(* IEC 61131-3 sources: com.logicals.lc3.webinar/usRTS_RPMControl_iSOC/src_FB_LIB_SAFE/Safe/PLCOpen, 23 files *)

(* ---- SF_MutingPar.iecst ---- *)
USING logicals.web.standard.safe;

NAMESPACE logicals.web.standard.safe
NAMESPACE plcopen

TYPE
	SF_MutingPar_State : UINT(
	/* Static Reset condition detected after FB activation in state 8401. */
	Reset_Error_1 := 16#C001,
	/* Static Reset condition detected in state 8402. */
	Reset_Error_2 := 16#C011,
	/* Error detected in muting sequence state 8000, 8010, 8310, 8020, 8040, 8030, 8330, 8110, 8410, 8120, 8140, 8130 or 8430. */
	Error_Muting_Sequence := 16#C004,
	/* DiscTime11_12, DiscTime21_22 or MaxMutingTime value out of range. */
	Parameter_Error := 16#C010,
	/* Timing error: Active muting time (when S_MutingActive = TRUE) exceeds MaxMutingTime. */
	Error_Timer_MaxMuting := 16#C020,
	/* Timing error: Discrepancy time for switching MutingSwitch11 and MutingSwitch12 > DiscTime11_12. */
	Error_Timer_MS11_12 := 16#C030,
	/* Timing error: Discrepancy time for switching MutingSwitch21 and MutingSwitch22 > DiscTime21_22. */
	Error_Timer_MS21_22 := 16#C040,
	/* Timing error: Discrepancy time for switching MutingSwitch21 and MutingSwitch22 > DiscTime21_22. */
	Idle := 16#0000,
	/* Muting not active and no safety demand from AOPD. If timers from subsequent muting are still running, they are stopped. */
	AOPD_Free := 16#8000,
	/* Function block has been activated. */
	Init := 16#8401,
	/* Safety demand detected by AOPD, muting not active. */
	Safety_Demand_AOPD := 16#8802,
	/* Safety demand or errors have been detected and are now cleared. Operator acknowledgment by Reset required. */
	Wait_for_Reset := 16#8402,
	/* Safety function activated. */
	Safe := 16#8002,
	/* Muting forward sequence is in starting phase after rising trigger of MutingSwitch 11.
	 * Monitoring of DiscTime11_12 is activated. Monitoring of MaxMutingTime is activated.
	 */
	Muting_Forward_Start_1 := 16#8010,
	/* Muting forward sequence is in starting phase after rising trigger of MutingSwitch 12. Monitoring of DiscTime11_12 is activated.
	 * Monitoring of MaxMutingTime is activated.
	 */
	Muting_Forward_Start_2 := 16#8310,
	/* Muting forward sequence is active either:
	 * - After rising trigger of the second entry MutingSwitch 12 or 11 has been detected.
	 * - When both MutingSwitch 11 and 12 have been actuated in the same cycle.
	 * Monitoring of DiscTime11_12 is stopped. Monitoring of MaxMutingTime is activated, when transition came directly from state 8000.
	 */
	Muting_Forward_Active_1 := 16#8020,
	/* Muting forward sequence is active. MutingSwitch21 is the first exit switch actuated. Monitoring of DiscTime21_22 is started. */
	Muting_Forward_Step_1 := 16#8030,
	/* Muting forward sequence is active. MutingSwitch22 is the first exit switch actuated. Monitoring of DiscTime21_22 is started. */
	Muting_Forward_Step_2 := 16#8330,
	/* Muting forward sequence is still active. Both MutingSwitch21 and 22 are actuated, the monitoring of DiscTime21_22 is stopped. */
	Muting_Forward_Active_2 := 16#8040,
	/* Muting backward sequence is in starting phase after rising trigger of MutingSwitch21.
	 * Monitoring of DiscTime21_22 is activated. Monitoring of MaxMutingTime is activated.
	 */
	Muting_Backward_Start_1 := 16#8110,
	/* Muting backward sequence is in starting phase after rising trigger of MutingSwitch22.
	 * Monitoring of DiscTime21_22 is activated. Monitoring of MaxMutingTime is activated.
	 */
	Muting_Backward_Start_2 := 16#8410,
	/* Muting backward sequence is active either:
	 * - After rising trigger of the second MutingSwitch 21 or 22 has been detected.
	 * - When both MutingSwitch 21 and 22 have been actuated in the same cycle.
	 * Monitoring of DiscTime21_22 is stopped. Monitoring of MaxMuting-Time is activated, when transition came directly from state 8000.
	 */
	Muting_Backward_Active_1 := 16#8120,
	/* Muting backward sequence is active. MutingSwitch11 is the first exit switch actuated. Monitoring of DiscTime11_12 is started. */
	Muting_Backward_Step_1 := 16#8130,
	/* Muting backward sequence is active. MutingSwitch12 is the first exit switch actuated. Monitoring of DiscTime11_12 is started. */
	Muting_Backward_Step_2 := 16#8430,
	/* Muting backward sequence is still active. Both exit switches MutingSwitch11 and 12 are actuated, the monitoring of DiscTime11_12 is stopped. */
	Muting_Backward_Active_2 := 16#8140
	);
END_TYPE

/* Muting is the intended suppression of the safety function. In this FB, parallel muting with four muting sensors is specified. */

FUNCTION_BLOCK SF_MutingPar
	{ altName:="SF_MutingPar"; bgColor:="Gold"; width:=360; }
	VAR_INPUT
		/* See Section 5.1.1 General Input Parameters */
		Activate : BOOL := FALSE;
		/* Variable.
		 * OSSD signal from AOPD.
		 * FALSE: Protection field interrupted.
		 * TRUE: Protection field not interrupted.
		 */
		S_AOPD_In : SAFEBOOL := SAFEBOOL_Constant#SAFEFALSE;
		/* Variable.
		 * Status of Muting sensor 11.
		 * FALSE: Muting sensor 11 not actuated.
		 * TRUE: Workpiece actuates muting sensor 11.
		 * Depending on the safety requirements it can be necessary to connect a SAFEBOOL.
		 */
		MutingSwitch11 : BOOL := FALSE;
		/* Variable.
		 * Status of Muting sensor 12.
		 * FALSE: Muting sensor 12 not actuated.
		 * TRUE: Workpiece actuates muting sensor 12.
		 * Depending on the safety requirements it can be necessary to connect a SAFEBOOL.
		 */
		MutingSwitch12 : BOOL := FALSE;
		/* Variable.
		 * Status of Muting sensor 21.
		 * FALSE: Muting sensor 21 not actuated.
		 * TRUE: Workpiece actuates muting sensor 21.
		 * Depending on the safety requirements it can be necessary to connect a SAFEBOOL.
		 */
		MutingSwitch21 : BOOL := FALSE;
		/* Variable.
		 * Status of Muting sensor 22.
		 * FALSE: Muting sensor 22 not actuated.
		 * TRUE: Workpiece actuates muting sensor 22.
		 * Depending on the safety requirements it can be necessary to connect a SAFEBOOL.
		 */
		MutingSwitch22 : BOOL := FALSE;
		/* Constant 0..4 s;
		 * Maximum discrepancy time for MutingSwitch11 and MutingSwitch12.
		 */
		DiscTime11_12 : TIME := T#0s;
		/* Constant 0..4 s;
		 * Maximum discrepancy time for MutingSwitch21 and MutingSwitch22.
		 */
		DiscTime21_22 : TIME := T#0s;
		/* Constant 0..120 min (application area specific);
		 * Maximum time for complete muting sequence, timer started when first 2 muting sensors are actuated.
		 */
		MaxMutingTime : TIME := T#0s;
		/* Variable or constant.
		 * Command by the control system that enables the start of the muting function when needed by the machine cycle.
		 * After the start of the muting function, this signal can be switched off.
		 * FALSE: Muting not enabled
		 * TRUE: Start of Muting function enabled
		 */
		MutingEnable : BOOL := FALSE;
		/* See Section 5.1.1 General Input Parameters */
		S_StartReset : SAFEBOOL := SAFEBOOL_Constant#SAFEFALSE;
		/* See Section 5.1.1 General Input Parameters */
		Reset : BOOL := FALSE;
	END_VAR
	VAR_OUTPUT
		/* See Section 5.1.2 General Output Parameters */
		Ready : BOOL := FALSE;
		/* Safety related output, indicates status of the muted guard.
		 * FALSE: AOPD protection field interrupted and muting not active.
		 * TRUE: AOPD protection field not interrupted or muting active.
		 */
		S_AOPD_Out : SAFEBOOL := SAFEBOOL_Constant#SAFEFALSE;
		/* Indicates status of Muting process.
		 * FALSE: Muting not active.
		 * TRUE: Muting active.
		 */
		S_MutingActive : SAFEBOOL := SAFEBOOL_Constant#SAFEFALSE;
		/* Optional. See 5.1.2 General Output Parameters */
		SafetyDemand : BOOL := FALSE;
		/* Optional. See 5.1.2 General Output Parameters */
		ResetRequest : BOOL := FALSE;
		/* See Section 5.1.2 General Output Parameters */
		Error : BOOL := FALSE;
		/* See Section 5.1.2 General Output Parameters */
		DiagCode : WORD := 16#000;
	END_VAR
	VAR
		/* ControlCode is used for state tracking */
		ControlCode : UINT := 16#0000;
		DiscTimer11_12 : TON;
		DiscTimer21_22 : TON;
		MaxMutingTimer : TON;
		R_Trig_Reset : R_TRIG;
		R_Trig_S11: R_TRIG;
		R_Trig_S12: R_TRIG;
		R_Trig_S21: R_TRIG;
		R_Trig_S22: R_TRIG;
		F_Trig_S11: F_TRIG;
		F_Trig_S12: F_TRIG;
		F_Trig_S21: F_TRIG;
		F_Trig_S22: F_TRIG;
	END_VAR

	R_Trig_Reset(Reset);
	R_Trig_S11(MutingSwitch11);
	R_Trig_S12(MutingSwitch12);
	R_Trig_S21(MutingSwitch21);
	R_Trig_S22(MutingSwitch22);
	F_Trig_S11(MutingSwitch11);
	F_Trig_S12(MutingSwitch12);
	F_Trig_S21(MutingSwitch21);
	F_Trig_S22(MutingSwitch22);

	IF(NOT Activate) THEN
		ControlCode := SF_MutingPar_State#Idle;
		DiagCode := TO_WORD(ControlCode);
	ELSE
		CASE TO_UINT(ControlCode) OF
			SF_MutingPar_State#Idle:
				/* IF(Activate) THEN - Active is always true here */
					ControlCode := SF_MutingPar_State#Init;
					DiagCode := TO_WORD(ControlCode);
			SF_MutingPar_State#Init:
				IF(Reset AND NOT R_Trig_Reset.Q) THEN
					ControlCode := SF_MutingPar_State#Reset_Error_1;
					DiagCode := TO_WORD(ControlCode);
				ELSIF(DiscTime11_12 > T#4s OR DiscTime11_12 < T#0s OR DiscTime21_22 > T#4s OR DiscTime21_22 < T#0s OR MaxMutingTime > T#120m OR MaxMutingTime < T#0m) THEN
					ControlCode := SF_MutingPar_State#Parameter_Error;
					DiagCode := TO_WORD(ControlCode);
				ELSIF(R_Trig_Reset.Q OR IS(S_StartReset)) THEN
					ControlCode := SF_MutingPar_State#Safe;
					DiagCode := TO_WORD(ControlCode);
				END_IF;
			SF_MutingPar_State#Reset_Error_1:
				IF(NOT Reset) THEN
					ControlCode := SF_MutingPar_State#Init;
					DiagCode := TO_WORD(ControlCode);
				END_IF;
			SF_MutingPar_State#Safe:
				IF(IS_NOT(S_AOPD_In)) THEN
					ControlCode := SF_MutingPar_State#Safety_Demand_AOPD;
					DiagCode := TO_WORD(ControlCode);
				/* ELSIF(IS(S_AOPD_In)) THEN */
				ELSE
					ControlCode := SF_MutingPar_State#AOPD_Free;
					DiagCode := TO_WORD(ControlCode);
				END_IF;
			SF_MutingPar_State#Safety_Demand_AOPD:
				IF(IS(S_AOPD_In)) THEN
					ControlCode := SF_MutingPar_State#Wait_for_Reset;
					DiagCode := TO_WORD(ControlCode);
				END_IF;
			SF_MutingPar_State#Wait_for_Reset:
				IF(Reset AND NOT R_Trig_Reset.Q) THEN
					ControlCode := SF_MutingPar_State#Reset_Error_2;
					DiagCode := TO_WORD(ControlCode);
				ELSIF(R_Trig_Reset.Q) THEN
					ControlCode := SF_MutingPar_State#Safe;
					DiagCode := TO_WORD(ControlCode);
				END_IF;
			SF_MutingPar_State#Reset_Error_2:
				IF(NOT Reset) THEN
					ControlCode := SF_MutingPar_State#Wait_for_Reset;
					DiagCode := TO_WORD(ControlCode);
				END_IF;
			SF_MutingPar_State#AOPD_Free:
				/* MutingEnable missing when muting sequence starts */
				IF(NOT MutingEnable) THEN
					IF((R_Trig_S11.Q AND NOT MutingSwitch12 AND NOT MutingSwitch21 AND NOT MutingSwitch22) OR
						(NOT MutingSwitch11 AND R_Trig_S12.Q AND NOT MutingSwitch21 AND NOT MutingSwitch22) OR
						(NOT MutingSwitch22 AND R_Trig_S21.Q AND NOT MutingSwitch11 AND NOT MutingSwitch12) OR
						(R_Trig_S22.Q AND NOT MutingSwitch21 AND NOT MutingSwitch11 AND NOT MutingSwitch12) OR
						(R_Trig_S11.Q AND R_Trig_S12.Q AND NOT MutingSwitch21 AND NOT MutingSwitch22) OR
						(R_Trig_S21.Q AND R_Trig_S22.Q AND NOT MutingSwitch11 AND NOT MutingSwitch12)) THEN
							ControlCode := SF_MutingPar_State#Error_Muting_Sequence;
							DiagCode := TO_WORD(SF_MutingPar_State#Error_Muting_Sequence + 16#0F00 + MutingParGetErrorStateOfMutingSensors(MutingSwitch11, MutingSwitch12, MutingSwitch21, MutingSwitch22));
					END_IF;
				/* wrong muting sequence */
				ELSIF((MutingSwitch11 OR MutingSwitch12) AND (MutingSwitch21 OR MutingSwitch22)) OR
					(R_Trig_S11.Q AND MutingSwitch12 AND NOT R_Trig_S12.Q) OR
					(R_Trig_S12.Q AND MutingSwitch11 AND NOT R_Trig_S11.Q) OR
					(R_Trig_S21.Q AND MutingSwitch22 AND NOT R_Trig_S22.Q) OR
					(R_Trig_S22.Q AND MutingSwitch21 AND NOT R_Trig_S21.Q) OR
					((MutingSwitch11 AND NOT R_Trig_S11.Q) AND (MutingSwitch12 AND NOT R_Trig_S12.Q)) OR
					((MutingSwitch21 AND NOT R_Trig_S21.Q) AND (MutingSwitch22 AND NOT R_Trig_S22.Q)) THEN
						ControlCode := SF_MutingPar_State#Error_Muting_Sequence;
						DiagCode := TO_WORD(SF_MutingPar_State#Error_Muting_Sequence + MutingParGetErrorStateOfMutingSensors(MutingSwitch11, MutingSwitch12, MutingSwitch21, MutingSwitch22));
				ELSIF(IS_NOT(S_AOPD_In)) THEN
					ControlCode := SF_MutingPar_State#Safety_Demand_AOPD;
					DiagCode := TO_WORD(ControlCode);
				ELSIF(MutingEnable AND (R_Trig_S11.Q AND NOT MutingSwitch12 AND NOT MutingSwitch21 AND NOT MutingSwitch22)) THEN
					ControlCode := SF_MutingPar_State#Muting_Forward_Start_1;
					DiagCode := TO_WORD(ControlCode);
				ELSIF(MutingEnable AND (NOT MutingSwitch11 AND R_Trig_S12.Q AND NOT MutingSwitch21 AND NOT MutingSwitch22)) THEN
					ControlCode := SF_MutingPar_State#Muting_Forward_Start_2;
					DiagCode := TO_WORD(ControlCode);
				ELSIF(MutingEnable AND (NOT MutingSwitch22 AND R_Trig_S21.Q AND NOT MutingSwitch11 AND NOT MutingSwitch12)) THEN
					ControlCode := SF_MutingPar_State#Muting_Backward_Start_1;
					DiagCode := TO_WORD(ControlCode);
				ELSIF(MutingEnable AND (R_Trig_S22.Q AND NOT MutingSwitch21 AND NOT MutingSwitch11 AND NOT MutingSwitch12)) THEN
					ControlCode := SF_MutingPar_State#Muting_Backward_Start_2;
					DiagCode := TO_WORD(ControlCode);
				ELSIF(MutingEnable AND (R_Trig_S11.Q AND R_Trig_S12.Q AND NOT MutingSwitch21 AND NOT MutingSwitch22)) THEN
					ControlCode := SF_MutingPar_State#Muting_Forward_Active_1;
					DiagCode := TO_WORD(ControlCode);
				ELSIF(MutingEnable AND (R_Trig_S21.Q AND R_Trig_S22.Q AND NOT MutingSwitch11 AND NOT MutingSwitch12)) THEN
					ControlCode := SF_MutingPar_State#Muting_Backward_Active_1;
					DiagCode := TO_WORD(ControlCode);
				END_IF;
			SF_MutingPar_State#Muting_Forward_Start_1:
				DiscTimer11_12();
				MaxMutingTimer();
				IF(NOT MutingEnable) THEN
					ControlCode := SF_MutingPar_State#Error_Muting_Sequence;
					DiagCode := TO_WORD(SF_MutingPar_State#Error_Muting_Sequence + 16#0F00 + MutingParGetErrorStateOfMutingSensors(MutingSwitch11, MutingSwitch12, MutingSwitch21, MutingSwitch22));
				ELSIF(NOT MutingSwitch11 OR MutingSwitch21 OR MutingSwitch22) THEN
					ControlCode := SF_MutingPar_State#Error_Muting_Sequence;
					DiagCode := TO_WORD(SF_MutingPar_State#Error_Muting_Sequence + 16#0100 + MutingParGetErrorStateOfMutingSensors(MutingSwitch11, MutingSwitch12, MutingSwitch21, MutingSwitch22));
				ELSIF(DiscTimer11_12.Q) THEN
					ControlCode := SF_MutingPar_State#Error_Timer_MS11_12;
					DiagCode := TO_WORD(ControlCode);
				ELSIF(MaxMutingTimer.Q) THEN
					ControlCode := SF_MutingPar_State#Error_Timer_MaxMuting;
					DiagCode := TO_WORD(ControlCode);
				ELSIF(IS_NOT(S_AOPD_In)) THEN
					ControlCode := SF_MutingPar_State#Safety_Demand_AOPD;
					DiagCode := TO_WORD(ControlCode);
				ELSIF(MutingEnable AND(MutingSwitch11 AND R_Trig_S12.Q AND NOT MutingSwitch21 AND NOT MutingSwitch22)) THEN
					ControlCode := SF_MutingPar_State#Muting_Forward_Active_1;
					DiagCode := TO_WORD(ControlCode);
				END_IF;
			SF_MutingPar_State#Muting_Forward_Start_2:
				DiscTimer11_12();
				MaxMutingTimer();
				IF(NOT MutingEnable) THEN
					ControlCode := SF_MutingPar_State#Error_Muting_Sequence;
					DiagCode := TO_WORD(SF_MutingPar_State#Error_Muting_Sequence + 16#0F00 + MutingParGetErrorStateOfMutingSensors(MutingSwitch11, MutingSwitch12, MutingSwitch21, MutingSwitch22));
				ELSIF(NOT MutingSwitch12 OR MutingSwitch21 OR MutingSwitch22) THEN
					ControlCode := SF_MutingPar_State#Error_Muting_Sequence;
					DiagCode := TO_WORD(SF_MutingPar_State#Error_Muting_Sequence + 16#0200 + MutingParGetErrorStateOfMutingSensors(MutingSwitch11, MutingSwitch12, MutingSwitch21, MutingSwitch22));
				ELSIF(DiscTimer11_12.Q) THEN
					ControlCode := SF_MutingPar_State#Error_Timer_MS11_12;
					DiagCode := TO_WORD(ControlCode);
				ELSIF(MaxMutingTimer.Q) THEN
					ControlCode := SF_MutingPar_State#Error_Timer_MaxMuting;
					DiagCode := TO_WORD(ControlCode);
				ELSIF(IS_NOT(S_AOPD_In)) THEN
					ControlCode := SF_MutingPar_State#Safety_Demand_AOPD;
					DiagCode := TO_WORD(ControlCode);
				ELSIF(R_Trig_S11.Q AND MutingSwitch12 AND NOT MutingSwitch21 AND NOT MutingSwitch22) THEN
					ControlCode := SF_MutingPar_State#Muting_Forward_Active_1;
					DiagCode := TO_WORD(ControlCode);
				END_IF;
			SF_MutingPar_State#Muting_Backward_Start_1:
				DiscTimer21_22();
				MaxMutingTimer();
				IF(NOT MutingEnable) THEN
					ControlCode := SF_MutingPar_State#Error_Muting_Sequence;
					DiagCode := TO_WORD(SF_MutingPar_State#Error_Muting_Sequence + 16#0F00 + MutingParGetErrorStateOfMutingSensors(MutingSwitch11, MutingSwitch12, MutingSwitch21, MutingSwitch22));
				ELSIF(MutingSwitch11 OR MutingSwitch12 OR NOT MutingSwitch21) THEN
					ControlCode := SF_MutingPar_State#Error_Muting_Sequence;
					DiagCode := TO_WORD(SF_MutingPar_State#Error_Muting_Sequence + 16#0700 + MutingParGetErrorStateOfMutingSensors(MutingSwitch11, MutingSwitch12, MutingSwitch21, MutingSwitch22));
				ELSIF(DiscTimer21_22.Q) THEN
					ControlCode := SF_MutingPar_State#Error_Timer_MS21_22;
					DiagCode := TO_WORD(ControlCode);
				ELSIF(MaxMutingTimer.Q) THEN
					ControlCode := SF_MutingPar_State#Error_Timer_MaxMuting;
					DiagCode := TO_WORD(ControlCode);
				ELSIF(IS_NOT(S_AOPD_In)) THEN
					ControlCode := SF_MutingPar_State#Safety_Demand_AOPD;
					DiagCode := TO_WORD(ControlCode);
				ELSIF(MutingEnable AND (MutingSwitch21 AND R_Trig_S22.Q AND NOT MutingSwitch11 AND NOT MutingSwitch12)) THEN
					ControlCode := SF_MutingPar_State#Muting_Backward_Active_1;
					DiagCode := TO_WORD(ControlCode);
				END_IF;
			SF_MutingPar_State#Muting_Backward_Start_2:
				DiscTimer21_22();
				MaxMutingTimer();
				IF(NOT MutingEnable) THEN
					ControlCode := SF_MutingPar_State#Error_Muting_Sequence;
					DiagCode := TO_WORD(SF_MutingPar_State#Error_Muting_Sequence + 16#0F00 + MutingParGetErrorStateOfMutingSensors(MutingSwitch11, MutingSwitch12, MutingSwitch21, MutingSwitch22));
				ELSIF(MutingSwitch11 OR MutingSwitch12 OR NOT MutingSwitch22) THEN
					ControlCode := SF_MutingPar_State#Error_Muting_Sequence;
					DiagCode := TO_WORD(SF_MutingPar_State#Error_Muting_Sequence + 16#0800 + MutingParGetErrorStateOfMutingSensors(MutingSwitch11, MutingSwitch12, MutingSwitch21, MutingSwitch22));
				ELSIF(DiscTimer21_22.Q) THEN
					ControlCode := SF_MutingPar_State#Error_Timer_MS21_22;
					DiagCode := TO_WORD(ControlCode);
				ELSIF(MaxMutingTimer.Q) THEN
					ControlCode := SF_MutingPar_State#Error_Timer_MaxMuting;
					DiagCode := TO_WORD(ControlCode);
				ELSIF(IS_NOT(S_AOPD_In)) THEN
					ControlCode := SF_MutingPar_State#Safety_Demand_AOPD;
					DiagCode := TO_WORD(ControlCode);
				ELSIF(MutingEnable AND (R_Trig_S21.Q AND MutingSwitch22 AND NOT MutingSwitch11 AND NOT MutingSwitch12)) THEN
					ControlCode := SF_MutingPar_State#Muting_Backward_Active_1;
					DiagCode := TO_WORD(ControlCode);
				END_IF;
			SF_MutingPar_State#Muting_Forward_Active_1:
				MaxMutingTimer();
				IF(NOT MutingSwitch11 OR NOT MutingSwitch12) THEN
					ControlCode := SF_MutingPar_State#Error_Muting_Sequence;
					DiagCode := TO_WORD(SF_MutingPar_State#Error_Muting_Sequence + 16#0300 + MutingParGetErrorStateOfMutingSensors(MutingSwitch11, MutingSwitch12, MutingSwitch21, MutingSwitch22));
				ELSIF(MaxMutingTimer.Q) THEN
					ControlCode := SF_MutingPar_State#Error_Timer_MaxMuting;
					DiagCode := TO_WORD(ControlCode);
				ELSIF(MutingSwitch11 AND MutingSwitch12 AND MutingSwitch21 AND MutingSwitch22) THEN
					ControlCode := SF_MutingPar_State#Muting_Forward_Active_2;
					DiagCode := TO_WORD(ControlCode);
				ELSIF(MutingSwitch11 AND MutingSwitch12 AND R_Trig_S21.Q AND NOT MutingSwitch22) THEN
					ControlCode := SF_MutingPar_State#Muting_Forward_Step_1;
					DiagCode := TO_WORD(ControlCode);
				ELSIF(MutingSwitch11 AND MutingSwitch12 AND NOT MutingSwitch21 AND R_Trig_S22.Q) THEN
					ControlCode := SF_MutingPar_State#Muting_Forward_Step_2;
					DiagCode := TO_WORD(ControlCode);
				END_IF;
			SF_MutingPar_State#Muting_Forward_Step_1:
				DiscTimer21_22();
				MaxMutingTimer();
				IF(NOT MutingSwitch11 OR NOT MutingSwitch12 OR NOT MutingSwitch21) THEN
					ControlCode := SF_MutingPar_State#Error_Muting_Sequence;
					DiagCode := TO_WORD(SF_MutingPar_State#Error_Muting_Sequence + 16#0400 + MutingParGetErrorStateOfMutingSensors(MutingSwitch11, MutingSwitch12, MutingSwitch21, MutingSwitch22));
				ELSIF(DiscTimer21_22.Q) THEN
					ControlCode := SF_MutingPar_State#Error_Timer_MS21_22;
					DiagCode := TO_WORD(ControlCode);
				ELSIF(MaxMutingTimer.Q) THEN
					ControlCode := SF_MutingPar_State#Error_Timer_MaxMuting;
					DiagCode := TO_WORD(ControlCode);
				ELSIF(MutingSwitch11 AND MutingSwitch12 AND MutingSwitch21 AND R_Trig_S22.Q) THEN
					ControlCode := SF_MutingPar_State#Muting_Forward_Active_2;
					DiagCode := TO_WORD(ControlCode);
				END_IF;
			SF_MutingPar_State#Muting_Forward_Step_2:
				DiscTimer21_22();
				MaxMutingTimer();
				IF(NOT MutingSwitch11 OR NOT MutingSwitch12 OR NOT MutingSwitch22) THEN
					ControlCode := SF_MutingPar_State#Error_Muting_Sequence;
					DiagCode := TO_WORD(SF_MutingPar_State#Error_Muting_Sequence + 16#0500 + MutingParGetErrorStateOfMutingSensors(MutingSwitch11, MutingSwitch12, MutingSwitch21, MutingSwitch22));
				ELSIF(DiscTimer21_22.Q) THEN
					ControlCode := SF_MutingPar_State#Error_Timer_MS21_22;
					DiagCode := TO_WORD(ControlCode);
				ELSIF(MaxMutingTimer.Q) THEN
					ControlCode := SF_MutingPar_State#Error_Timer_MaxMuting;
					DiagCode := TO_WORD(ControlCode);
				ELSIF(MutingSwitch11 AND MutingSwitch12 AND R_Trig_S21.Q AND MutingSwitch22) THEN
					ControlCode := SF_MutingPar_State#Muting_Forward_Active_2;
					DiagCode := TO_WORD(ControlCode);
				END_IF;
			SF_MutingPar_State#Muting_Forward_Active_2:
				MaxMutingTimer();
				IF(R_Trig_S11.Q OR R_Trig_S12.Q OR R_Trig_S21.Q OR R_Trig_S22.Q) OR
					((MutingSwitch11 OR MutingSwitch12) AND (F_Trig_S21.Q OR F_Trig_S22.Q)) OR
					((F_Trig_S11.Q OR F_Trig_S12.Q) AND (F_Trig_S21.Q OR F_Trig_S22.Q)) THEN
						ControlCode := SF_MutingPar_State#Error_Muting_Sequence;
						DiagCode := TO_WORD(SF_MutingPar_State#Error_Muting_Sequence + 16#0600 + MutingParGetErrorStateOfMutingSensors(MutingSwitch11, MutingSwitch12, MutingSwitch21, MutingSwitch22));
				ELSIF(MaxMutingTimer.Q) THEN
					ControlCode := SF_MutingPar_State#Error_Timer_MaxMuting;
					DiagCode := TO_WORD(ControlCode);
				ELSIF(NOT MutingSwitch11 AND NOT MutingSwitch12) AND (F_Trig_S21.Q OR F_Trig_S22.Q) THEN
					ControlCode := SF_MutingPar_State#AOPD_Free;
					DiagCode := TO_WORD(ControlCode);
				END_IF;
			SF_MutingPar_State#Muting_Backward_Active_1:
				MaxMutingTimer();
				IF(NOT MutingSwitch21 OR NOT MutingSwitch22) THEN
					ControlCode := SF_MutingPar_State#Error_Muting_Sequence;
					DiagCode := TO_WORD(SF_MutingPar_State#Error_Muting_Sequence + 16#0900 + MutingParGetErrorStateOfMutingSensors(MutingSwitch11, MutingSwitch12, MutingSwitch21, MutingSwitch22));
				ELSIF(MaxMutingTimer.Q) THEN
					ControlCode := SF_MutingPar_State#Error_Timer_MaxMuting;
					DiagCode := TO_WORD(ControlCode);
				ELSIF(MutingSwitch11 AND MutingSwitch12 AND MutingSwitch21 AND MutingSwitch22) THEN
					ControlCode := SF_MutingPar_State#Muting_Backward_Active_2;
					DiagCode := TO_WORD(ControlCode);
				ELSIF(MutingSwitch21 AND MutingSwitch22 AND R_Trig_S11.Q AND NOT MutingSwitch12) THEN
					ControlCode := SF_MutingPar_State#Muting_Backward_Step_1;
					DiagCode := TO_WORD(ControlCode);
				ELSIF(MutingSwitch21 AND MutingSwitch22 AND NOT MutingSwitch11 AND R_Trig_S12.Q) THEN
					ControlCode := SF_MutingPar_State#Muting_Backward_Step_2;
					DiagCode := TO_WORD(ControlCode);
				END_IF;
			SF_MutingPar_State#Muting_Backward_Step_1:
				MaxMutingTimer();
				DiscTimer11_12();
				IF(NOT MutingSwitch21 OR NOT MutingSwitch22 OR NOT MutingSwitch11) THEN
					ControlCode := SF_MutingPar_State#Error_Muting_Sequence;
					DiagCode := TO_WORD(SF_MutingPar_State#Error_Muting_Sequence + 16#0A00 + MutingParGetErrorStateOfMutingSensors(MutingSwitch11, MutingSwitch12, MutingSwitch21, MutingSwitch22));
				ELSIF(DiscTimer11_12.Q) THEN
					ControlCode := SF_MutingPar_State#Error_Timer_MS11_12;
					DiagCode := TO_WORD(ControlCode);
				ELSIF(MaxMutingTimer.Q) THEN
					ControlCode := SF_MutingPar_State#Error_Timer_MaxMuting;
					DiagCode := TO_WORD(ControlCode);
				ELSIF(MutingSwitch21 AND MutingSwitch22 AND MutingSwitch11 AND R_Trig_S12.Q) THEN
					ControlCode := SF_MutingPar_State#Muting_Backward_Active_2;
					DiagCode := TO_WORD(ControlCode);
				END_IF;
			SF_MutingPar_State#Muting_Backward_Step_2:
				MaxMutingTimer();
				DiscTimer11_12();
				IF(NOT MutingSwitch21 OR NOT MutingSwitch22 OR NOT MutingSwitch12) THEN
					ControlCode := SF_MutingPar_State#Error_Muting_Sequence;
					DiagCode := TO_WORD(SF_MutingPar_State#Error_Muting_Sequence + 16#0B00 + MutingParGetErrorStateOfMutingSensors(MutingSwitch11, MutingSwitch12, MutingSwitch21, MutingSwitch22));
				ELSIF(DiscTimer11_12.Q) THEN
					ControlCode := SF_MutingPar_State#Error_Timer_MS11_12;
					DiagCode := TO_WORD(ControlCode);
				ELSIF(MaxMutingTimer.Q) THEN
					ControlCode := SF_MutingPar_State#Error_Timer_MaxMuting;
					DiagCode := TO_WORD(ControlCode);
				ELSIF(MutingSwitch21 AND MutingSwitch22 AND R_Trig_S11.Q AND MutingSwitch12) THEN
					ControlCode := SF_MutingPar_State#Muting_Backward_Active_2;
					DiagCode := TO_WORD(ControlCode);
				END_IF;
			SF_MutingPar_State#Muting_Backward_Active_2:
				MaxMutingTimer();
				IF(R_Trig_S11.Q OR R_Trig_S12.Q OR R_Trig_S21.Q OR R_Trig_S22.Q) OR
					((MutingSwitch21 OR MutingSwitch22) AND (F_Trig_S11.Q OR F_Trig_S12.Q)) OR
					((F_Trig_S11.Q OR F_Trig_S12.Q) AND (F_Trig_S21.Q OR F_Trig_S22.Q)) THEN
						ControlCode := SF_MutingPar_State#Error_Muting_Sequence;
						DiagCode := TO_WORD(SF_MutingPar_State#Error_Muting_Sequence + 16#0C00 + MutingParGetErrorStateOfMutingSensors(MutingSwitch11, MutingSwitch12, MutingSwitch21, MutingSwitch22));
				ELSIF(MaxMutingTimer.Q) THEN
					ControlCode := SF_MutingPar_State#Error_Timer_MaxMuting;
					DiagCode := TO_WORD(ControlCode);
				ELSIF(NOT MutingSwitch21 AND NOT MutingSwitch22 AND(F_Trig_S11.Q OR F_Trig_S12.Q)) THEN
					ControlCode := SF_MutingPar_State#AOPD_Free;
					DiagCode := TO_WORD(ControlCode);
				END_IF;
			SF_MutingPar_State#Error_Timer_MaxMuting,
			SF_MutingPar_State#Error_Timer_MS11_12,
			SF_MutingPar_State#Error_Timer_MS21_22:
				IF(NOT(MutingSwitch11 OR MutingSwitch12 OR MutingSwitch21 OR MutingSwitch22)) THEN
					ControlCode := SF_MutingPar_State#Wait_for_Reset;
					DiagCode := TO_WORD(ControlCode);
				END_IF;
			ELSE
				ENO := FALSE;
		END_CASE;
	END_IF;

	CASE TO_UINT(ControlCode) OF
		SF_MutingPar_State#Reset_Error_1,
		SF_MutingPar_State#Reset_Error_2,
		SF_MutingPar_State#Parameter_Error,
		SF_MutingPar_State#Error_Timer_MaxMuting,
		SF_MutingPar_State#Error_Timer_MS11_12,
		SF_MutingPar_State#Error_Timer_MS21_22:
			DiscTimer11_12(IN := FALSE);
			DiscTimer21_22(IN := FALSE);
			MaxMutingTimer(IN := FALSE);
			Ready := TRUE;
			S_AOPD_Out := SAFEBOOL_Constant#SAFEFALSE;
			S_MutingActive := SAFEBOOL_Constant#SAFEFALSE;
			SafetyDemand := FALSE;
			ResetRequest := FALSE;
			Error := TRUE;
		SF_MutingPar_State#Error_Muting_Sequence:
			DiscTimer11_12(IN := FALSE);
			DiscTimer21_22(IN := FALSE);
			MaxMutingTimer(IN := FALSE);
			Ready := TRUE;
			S_AOPD_Out := SAFEBOOL_Constant#SAFEFALSE;
			S_MutingActive := SAFEBOOL_Constant#SAFEFALSE;
			SafetyDemand := FALSE;
			ResetRequest := FALSE;
			Error := TRUE;
		SF_MutingPar_State#Idle:
			DiscTimer11_12(IN := FALSE);
			DiscTimer21_22(IN := FALSE);
			MaxMutingTimer(IN := FALSE);
			Ready := FALSE;
			S_AOPD_Out := SAFEBOOL_Constant#SAFEFALSE;
			S_MutingActive := SAFEBOOL_Constant#SAFEFALSE;
			SafetyDemand := FALSE;
			ResetRequest := FALSE;
			Error := FALSE;
		SF_MutingPar_State#AOPD_Free:
			DiscTimer11_12(IN := FALSE);
			DiscTimer21_22(IN := FALSE);
			MaxMutingTimer(IN := FALSE);
			Ready := TRUE;
			S_AOPD_Out := SAFEBOOL_Constant#SAFETRUE;
			S_MutingActive := SAFEBOOL_Constant#SAFEFALSE;
			SafetyDemand := FALSE;
			ResetRequest := FALSE;
			Error := FALSE;
		SF_MutingPar_State#Muting_Forward_Start_1,
		SF_MutingPar_State#Muting_Forward_Start_2:
			DiscTimer11_12(IN := TRUE, PT := DiscTime11_12);
			DiscTimer21_22(IN := FALSE);
			MaxMutingTimer(IN := TRUE, PT := MaxMutingTime);
			Ready := TRUE;
			S_AOPD_Out := SAFEBOOL_Constant#SAFETRUE;
			S_MutingActive := SAFEBOOL_Constant#SAFEFALSE;
			SafetyDemand := FALSE;
			ResetRequest := FALSE;
			Error := FALSE;
		SF_MutingPar_State#Muting_Backward_Start_1,
		SF_MutingPar_State#Muting_Backward_Start_2:
			DiscTimer11_12(IN := FALSE);
			DiscTimer21_22(IN := TRUE, PT := DiscTime21_22);
			MaxMutingTimer(IN := TRUE, PT := MaxMutingTime);
			Ready := TRUE;
			S_AOPD_Out := SAFEBOOL_Constant#SAFETRUE;
			S_MutingActive := SAFEBOOL_Constant#SAFEFALSE;
			SafetyDemand := FALSE;
			ResetRequest := FALSE;
			Error := FALSE;
		SF_MutingPar_State#Init,
		SF_MutingPar_State#Wait_for_Reset:
			DiscTimer11_12(IN := FALSE);
			DiscTimer21_22(IN := FALSE);
			MaxMutingTimer(IN := FALSE);
			Ready := TRUE;
			S_AOPD_Out := SAFEBOOL_Constant#SAFEFALSE;
			S_MutingActive := SAFEBOOL_Constant#SAFEFALSE;
			SafetyDemand := FALSE;
			ResetRequest := TRUE;
			Error := FALSE;
		SF_MutingPar_State#Safety_Demand_AOPD:
			DiscTimer11_12(IN := FALSE);
			DiscTimer21_22(IN := FALSE);
			MaxMutingTimer(IN := FALSE);
			Ready := TRUE;
			S_AOPD_Out := SAFEBOOL_Constant#SAFEFALSE;
			S_MutingActive := SAFEBOOL_Constant#SAFEFALSE;
			SafetyDemand := TRUE;
			ResetRequest := FALSE;
			Error := FALSE;
		SF_MutingPar_State#Safe:
			DiscTimer11_12(IN := FALSE);
			DiscTimer21_22(IN := FALSE);
			MaxMutingTimer(IN := FALSE);
			Ready := TRUE;
			S_AOPD_Out := SAFEBOOL_Constant#SAFEFALSE;
			S_MutingActive := SAFEBOOL_Constant#SAFEFALSE;
			SafetyDemand := FALSE;
			ResetRequest := FALSE;
			Error := FALSE;
		SF_MutingPar_State#Muting_Backward_Active_1:
			DiscTimer11_12(IN := FALSE);
			DiscTimer21_22(IN := FALSE);
			IF(MutingEnable AND (R_Trig_S21.Q AND R_Trig_S22.Q AND NOT MutingSwitch11 AND NOT MutingSwitch12)) THEN
				MaxMutingTimer(IN := TRUE, PT:= MaxMutingTime);
			END_IF;
			Ready := TRUE;
			S_AOPD_Out := SAFEBOOL_Constant#SAFETRUE;
			S_MutingActive := SAFEBOOL_Constant#SAFETRUE;
			SafetyDemand := FALSE;
			ResetRequest := FALSE;
			Error := FALSE;
		SF_MutingPar_State#Muting_Backward_Step_1,
		SF_MutingPar_State#Muting_Backward_Step_2:
			DiscTimer11_12(IN := TRUE, PT := DiscTime11_12);
			DiscTimer21_22(IN := FALSE);
			Ready := TRUE;
			S_AOPD_Out := SAFEBOOL_Constant#SAFETRUE;
			S_MutingActive := SAFEBOOL_Constant#SAFETRUE;
			SafetyDemand := FALSE;
			ResetRequest := FALSE;
			Error := FALSE;
		SF_MutingPar_State#Muting_Backward_Active_2:
			DiscTimer11_12(IN := FALSE);
			DiscTimer21_22(IN := FALSE);
			Ready := TRUE;
			S_AOPD_Out := SAFEBOOL_Constant#SAFETRUE;
			S_MutingActive := SAFEBOOL_Constant#SAFETRUE;
			SafetyDemand := FALSE;
			ResetRequest := FALSE;
			Error := FALSE;
		SF_MutingPar_State#Muting_Forward_Active_1:
			DiscTimer11_12(IN := FALSE);
			DiscTimer21_22(IN := FALSE);
			IF(MutingEnable AND (R_Trig_S11.Q AND R_Trig_S12.Q AND NOT MutingSwitch21 AND NOT MutingSwitch22)) THEN
				MaxMutingTimer(IN := TRUE, PT:= MaxMutingTime);
			END_IF;
			Ready := TRUE;
			S_AOPD_Out := SAFEBOOL_Constant#SAFETRUE;
			S_MutingActive := SAFEBOOL_Constant#SAFETRUE;
			SafetyDemand := FALSE;
			ResetRequest := FALSE;
			Error := FALSE;
		SF_MutingPar_State#Muting_Forward_Step_1,
		SF_MutingPar_State#Muting_Forward_Step_2:
			DiscTimer11_12(IN := FALSE);
			DiscTimer21_22(IN := TRUE, PT := DiscTime21_22);
			Ready := TRUE;
			S_AOPD_Out := SAFEBOOL_Constant#SAFETRUE;
			S_MutingActive := SAFEBOOL_Constant#SAFETRUE;
			SafetyDemand := FALSE;
			ResetRequest := FALSE;
			Error := FALSE;
		SF_MutingPar_State#Muting_Forward_Active_2:
			DiscTimer11_12(IN := FALSE);
			DiscTimer21_22(IN := FALSE);
			Ready := TRUE;
			S_AOPD_Out := SAFEBOOL_Constant#SAFETRUE;
			S_MutingActive := SAFEBOOL_Constant#SAFETRUE;
			SafetyDemand := FALSE;
			ResetRequest := FALSE;
			Error := FALSE;
		ELSE
			ENO := FALSE;
	END_CASE;

	ENO := ENO AND CheckSAFEBOOL(S_AOPD_In) AND CheckSAFEBOOL(S_StartReset);

END_FUNCTION_BLOCK

FUNCTION MutingParGetErrorStateOfMutingSensors : UINT
	VAR_INPUT
		MS_11 : BOOL;
		MS_12 : BOOL;
		MS_21 : BOOL;
		MS_22 : BOOL;
	END_VAR

	VAR
		Result : UINT;
	END_VAR

	IF(MS_11) THEN
		Result := Result + 16#0010;
	END_IF;
	IF(MS_12) THEN
		Result := Result + 16#0020;
	END_IF;
	IF(MS_21) THEN
		Result := Result + 16#0040;
	END_IF;
	IF(MS_22) THEN
		Result := Result + 16#0080;
	END_IF;

	MutingParGetErrorStateOfMutingSensors := Result;

END_FUNCTION

END_NAMESPACE
END_NAMESPACE

(* ---- SF_Antivalent.iecst ---- *)
USING logicals.web.standard.safe;

NAMESPACE logicals.web.standard.safe
NAMESPACE plcopen

TYPE
	SF_Antivalent_State : UINT(
	/* Discrepancy time elapsed in state 8802. */
	Error_1 := 16#C010,
	/* Discrepancy time elapsed in state 8804. */
	Error_2 := 16#C020,
	/* Discrepancy time elapsed in state 8806. */
	Error_3 := 16#C030,
	/* The function block is not active (initial state). */
	Idle := 16#0000,
	/* An activation has been detected by the FB and the FB is now activated. */
	Init := 16#8801,
	/* The inputs switched to the Active state in antivalent mode. */
	Safety_Output_Enabled := 16#8000,
	/* ChannelNC has been switched to TRUE - waiting for ChannelNO to be switched to FALSE; discrepancy timer started. */
	Wait_for_NO := 16#8802,
	/* ChannelNO has been switched to FALSE - waiting for ChannelNC to be switched to TRUE; discrepancy timer started. */
	Wait_for_NC := 16#8804,
	/* One channel has been switched to inactive; waiting for the second channel to be switched to inactive too. */
	From_Active_Wait := 16#8806
	);
END_TYPE

/*
 * This function block converts two antivalent SAFEBOOL inputs (NO/NC pair) to one SAFEBOOL output with discrepancy time monitoring.
 * This FB should not be used stand-alone since it has no restart interlock.
 * It is required to connect the output to other safety related functionalities.
 */
FUNCTION_BLOCK SF_Antivalent
	{ altName:="SF_Antivalent"; bgColor:="Gold"; width:=380; }
	VAR_INPUT
		/* See Section 5.1.1 General Input Parameters */
		Activate : BOOL := FALSE;
		/* Variable. NC stands for Normally Closed.
		 * Input for NC connection.
		 * FALSE: NC contact open.
		 * TRUE: NC contact closed. */
		S_ChannelNC : SAFEBOOL := SAFEBOOL_Constant#SAFEFALSE;
		/* Variable. NO stands for Normally Open.
		 * Input for NO connection.
		 * FALSE: NO contact open
		 * TRUE: NO contact closed */
		S_ChannelNO : SAFEBOOL := SAFEBOOL_Constant#SAFETRUE;
		/* Constant. Maximum monitoring time for discrepancy status of both inputs. */
		DiscrepancyTime : TIME := T#0ms;
	END_VAR
	VAR_OUTPUT
		/* See Section 5.1.2 General Output Parameters */
		Ready : BOOL := FALSE;
		/* Safety related output
		 * FALSE: Minimum of one input signal "not active" or status change outside of monitoring time.
		 * TRUE: Both inputs signals "active" and status change within monitoring time. */
		S_AntivalentOut : SAFEBOOL := SAFEBOOL_Constant#SAFEFALSE;
		/* See 5.1.2 General Output Parameters */
		SafetyDemand : BOOL := FALSE;
		/* See Section 5.1.2 General Output Parameters */
		Error : BOOL := FALSE;
		/* See Section 5.1.2 General Output Parameters */
		DiagCode : WORD := 16#0000;
	END_VAR
	VAR
		DiscrepancyTimer : TON;
	END_VAR

	IF(NOT Activate) THEN
		DiagCode := TO_WORD(SF_Antivalent_State#Idle);
	ELSE
		CASE TO_UINT(DiagCode) OF
			SF_Antivalent_State#Idle:
				/* IF(Activate) THEN - Active is always true here */
					DiagCode := TO_WORD(SF_Antivalent_State#Init);
			SF_Antivalent_State#Init:
				IF(IS(S_ChannelNC) AND IS(S_ChannelNO)) THEN
					DiagCode := TO_WORD(SF_Antivalent_State#Wait_for_NO);
				ELSIF(IS_NOT(S_ChannelNC) AND IS_NOT(S_ChannelNO)) THEN
					DiagCode := TO_WORD(SF_Antivalent_State#Wait_for_NC);
				ELSIF(IS(S_ChannelNC) AND IS_NOT(S_ChannelNO)) THEN
					DiagCode := TO_WORD(SF_Antivalent_State#Safety_Output_Enabled);
				END_IF;
			SF_Antivalent_State#Wait_for_NO:
				DiscrepancyTimer();
				IF(DiscrepancyTimer.Q) THEN
					DiagCode := TO_WORD(SF_Antivalent_State#Error_1);
				ELSIF(IS_NOT(S_ChannelNC)) THEN
					DiagCode := TO_WORD(SF_Antivalent_State#Init);
				ELSIF(IS_NOT(S_ChannelNO)) THEN
					DiagCode := TO_WORD(SF_Antivalent_State#Safety_Output_Enabled);
				END_IF;
			SF_Antivalent_State#Wait_for_NC:
				DiscrepancyTimer();
				IF(DiscrepancyTimer.Q) THEN
					DiagCode := TO_WORD(SF_Antivalent_State#Error_2);
				ELSIF(IS(S_ChannelNO)) THEN
					DiagCode := TO_WORD(SF_Antivalent_State#Init);
				ELSIF(IS(S_ChannelNC)) THEN
					DiagCode := TO_WORD(SF_Antivalent_State#Safety_Output_Enabled);
				END_IF;
			SF_Antivalent_State#Safety_Output_Enabled:
				IF(IS_NOT(S_ChannelNC) AND IS(S_ChannelNO)) THEN
					DiagCode := TO_WORD(SF_Antivalent_State#Init);
				ELSIF(IS_NOT(S_ChannelNC) OR IS(S_ChannelNO)) THEN
					DiagCode := TO_WORD(SF_Antivalent_State#From_Active_Wait);
				END_IF;
			SF_Antivalent_State#From_Active_Wait:
				DiscrepancyTimer();
				IF(DiscrepancyTimer.Q) THEN
					DiagCode := TO_WORD(SF_Antivalent_State#Error_3);
				ELSIF(IS_NOT(S_ChannelNC) AND IS(S_ChannelNO)) THEN
					DiagCode := TO_WORD(SF_Antivalent_State#Init);
				END_IF;
			SF_Antivalent_State#Error_1,SF_Antivalent_State#Error_2,SF_Antivalent_State#Error_3:
				IF(IS_NOT(S_ChannelNC) AND IS(S_ChannelNO)) THEN
					DiagCode := TO_WORD(SF_Antivalent_State#Init);
				END_IF;
			ELSE
				ENO := FALSE;
		END_CASE;
	END_IF;

	CASE TO_UINT(DiagCode) OF
		SF_Antivalent_State#Idle:
			DiscrepancyTimer(IN := FALSE);
			Ready := FALSE;
			S_AntivalentOut := SAFEBOOL_Constant#SAFEFALSE;
			SafetyDemand := FALSE;
			Error := FALSE;
		SF_Antivalent_State#Init:
			DiscrepancyTimer(IN := FALSE);
			Ready := TRUE;
			S_AntivalentOut := SAFEBOOL_Constant#SAFEFALSE;
			SafetyDemand := TRUE;
			Error := FALSE;
		SF_Antivalent_State#Safety_Output_Enabled:
			DiscrepancyTimer(IN := FALSE);
			Ready := TRUE;
			S_AntivalentOut := SAFEBOOL_Constant#SAFETRUE;
			SafetyDemand := FALSE;
			Error := FALSE;
		SF_Antivalent_State#Wait_for_NO,SF_Antivalent_State#Wait_for_NC,SF_Antivalent_State#From_Active_Wait:
			DiscrepancyTimer(IN := TRUE, PT := DiscrepancyTime);
			Ready := TRUE;
			S_AntivalentOut := SAFEBOOL_Constant#SAFEFALSE;
			SafetyDemand := TRUE;
			Error := FALSE;
		SF_Antivalent_State#Error_1,SF_Antivalent_State#Error_2,SF_Antivalent_State#Error_3:
			DiscrepancyTimer(IN := FALSE);
			Ready := TRUE;
			S_AntivalentOut := SAFEBOOL_Constant#SAFEFALSE;
			SafetyDemand := FALSE;
			Error := TRUE;
		ELSE
			ENO := FALSE;
	END_CASE;

	ENO := ENO AND CheckSAFEBOOL(S_ChannelNC) AND CheckSAFEBOOL(S_ChannelNO);

END_FUNCTION_BLOCK

END_NAMESPACE
END_NAMESPACE

(* ---- SF_EDM.iecst ---- *)
USING logicals.web.standard.safe;

NAMESPACE logicals.web.standard.safe
NAMESPACE plcopen

TYPE

	SF_EDM_State : UINT(
	/* Static Reset signal in state 8001. */
	Reset_Error_1 := 16#C001,
	/* Static Reset signal or same signals at EDM1 and Reset (rising trigger at Reset and EDM1 at the same time) in state C010. */
	Reset_Error_21 := 16#C011,
	/* Static Reset signal or same signals at EDM2 and Reset (rising trigger at Reset and EDM2 at the same time) in state C020. */
	Reset_Error_22 := 16#C021,
	/* Static Reset signal or same signals at EDM1, EDM2, and Reset (rising trigger at Reset, EDM1, and EDM2 at the same time) in state C030. */
	Reset_Error_23 := 16#C031,
	/* Static Reset signal or same signals at EDM1 and Reset (rising trigger at Reset and EDM1 at the same time) in state C040. */
	Reset_Error_31 := 16#C041,
	/* Static Reset signal or same signals at EDM2 and Reset (rising trigger at Reset and EDM2 at the same time) in state C050. */
	Reset_Error_32 := 16#C051,
	/* Static Reset signal or same signals at EDM1, EDM2, and Reset (rising trigger at Reset, EDM1, and EDM2 at the same time) in state C060. */
	Reset_Error_33 := 16#C061,
	/* Static Reset signal in state C070. */
	Reset_Error_41 := 16#C071,
	/* Static Reset signal in state C080. */
	Reset_Error_42 := 16#C081,
	/* Static Reset signal in state C090. */
	Reset_Error_43 := 16#C091,

	/* The signal at EDM1 is not valid in the initial actuator state. In state 8010 the EDM1 signal is FALSE when enabling O_OutControl. */
	EDM_Error_11 := 16#C010,
	/* The signal at EDM2 is not valid in the initial actuator state. In state 8010 the EDM2 signal is FALSE when enabling O_OutControl. */
	EDM_Error_12 := 16#C020,
	/* The signals at EDM1 and EDM2 are not valid in the initial actuator states. In state 8010 the EDM1 and EDM2 signals are FALSE when ena-bling O_OutControl. */
	EDM_Error_13 := 16#C030,
	/* The signal at EDM1 is not valid in the initial actuator state. In state 8010 the EDM1 signal is FALSE and the monitoring time has elapsed. */
	EDM_Error_21 := 16#C040,
	/* The signal at EDM2 is not valid in the initial actuator state. In state 8010 the EDM2 signal is FALSE and the monitoring time has elapsed. */
	EDM_Error_22 := 16#C050,
	/* The signals at EDM1 and EDM2 are not valid in the initial actuator states. In state 8010 the EDM1 and EDM2 signals are FALSE and the monitoring time has elapsed. */
	EDM_Error_23 := 16#C060,
	/* The signal at EDM1 is not valid in the actuator switching state. In state 8000 the EDM1 signal is TRUE and the monitoring time has elapsed. */
	EDM_Error_31 := 16#C070,
	/* The signal at EDM2 is not valid in the actuator switching state. In state 8000 the EDM2 signal is TRUE and the monitoring time has elapsed. */
	EDM_Error_32 := 16#C080,
	/* The signals at EDM1 and EDM2 are not valid in the actuator switching state. In state 8000 the EDM1 and EDM2 signals are TRUE and the monitoring time has elapsed. */
	EDM_Error_33 := 16#C090,
	/* Similar signals at S_OutControl and Reset (R_TRIG at same cycle) de-tected (may be a programming error) */
	Init_Error := 16#C100,
	/* The function block is not active (initial state). */
	Idle := 16#0000,
	/* Block activation startup inhibit is active. Reset required. */
	Init := 16#8401,
	/* EDM control is not active. Timer starts when state is entered */
	Output_Disable := 16#8802,
	/* EDM control is active. Timer starts when state is entered */
	Output_Enable := 16#8000
	);

END_TYPE

/* External device monitoring - The FB controls a safety output and monitors controlled actuators, e.g. subsequent contactors */
FUNCTION_BLOCK SF_EDM
	{ altName:="SF_EDM"; bgColor:="Gold"; width:=320; }

	VAR_INPUT
		/* See Section 5.1.1 General Input Parameters */
		Activate : BOOL := FALSE;
		/* Variable.
		 * Control signal of the preceeding safety FB's.
		 * Typical function block signals from the library
		 * (e.g., SF_OutControl, SF_TwoHandControlTypeII, and/or others).
		 * FALSE: Disable safety output (S_EDM_Out).
		 * TRUE: Enable safety output (S_EDM_Out). */
		S_OutControl : SAFEBOOL := SAFEBOOL_Constant#SAFEFALSE;
		/* Variable.
		 * Feedback signal of the first connected actuator.
		 * FALSE: Switching state of the first connected actuator.
		 * TRUE: Initial state of the first connected actuator. */
		EDM1 : BOOL := FALSE;
		/* Variable.
		 * Feedback signal of the second connected actuator.
		 * According to the actuators installed, the wiring between the feedback signals and the targeted safety level, it can be that only combined input is used here. In that case the user must use a graphic connection to jumper the EDM1 and EDM2 parameters. EDM1 and EDM2 are then con-trolled by the same signal.
		 * FALSE: Switching state of the second connected actuator.
		 * TRUE: Initial state of the second connected actuator. */
		EDM2 : BOOL := FALSE;
		/* Constant.
		 * Max. response time of the connected and monitored actuators. */
		MonitoringTime : TIME := T#0ms;
		/* See Section 5.1.1 General Input Parameters */
		Reset : BOOL := FALSE;
	END_VAR

	VAR_OUTPUT
		/* See Section 5.1.2 General Output Parameters */
		Ready : BOOL := FALSE;
		/* Controls the actuator. The result is monitored by the feedback signal EDMx.
		 * FALSE: Disable connected actuators.
		 * TRUE: Enable connected actuators. */
		S_EDM_Out : SAFEBOOL := SAFEBOOL_Constant#SAFEFALSE;
		/* See Section 5.1.2 General Output Parameters */
		SafetyDemand : BOOL := FALSE;
		/* See Section 5.1.2 General Output Parameters */
		ResetRequest : BOOL := FALSE;
		/* See Section 5.1.2 General Output Parameters */
		Error : BOOL := FALSE;
		/* See Section 5.1.2 General Output Parameters */
		DiagCode : WORD := 16#0000;
	END_VAR

	VAR
		R_Trig_Reset : R_TRIG;
		R_Trig_S_OutControl : R_TRIG;
		R_Trig_EDM1 : R_TRIG;
		R_Trig_EDM2 : R_TRIG;
		MonitoringTimer_OutputDisable : TON;
		MonitoringTimer_OutputEnable : TON;
	END_VAR

	R_Trig_Reset(Reset);
	R_Trig_EDM1(EDM1);
	R_Trig_EDM2(EDM2);
	R_Trig_S_OutControl(IS(S_OutControl));

	IF(NOT Activate) THEN
		DiagCode := TO_WORD(SF_EDM_State#Idle);
	ELSE
		CASE TO_UINT(DiagCode) OF
			SF_EDM_State#Idle:
				/* IF(Activate) THEN - Activate is always true here */
					DiagCode := TO_WORD(SF_EDM_State#Init);
			SF_EDM_State#Init:
				IF(Reset AND NOT R_Trig_Reset.Q) THEN
					DiagCode := TO_WORD(SF_EDM_State#Reset_Error_1);
				ELSIF(R_Trig_Reset.Q AND R_Trig_S_OutControl.Q) THEN
					DiagCode := TO_WORD(SF_EDM_State#Init_Error);
				ELSIF(R_Trig_Reset.Q) THEN
					DiagCode := TO_WORD(SF_EDM_State#Output_Disable);
				END_IF;
			SF_EDM_State#Reset_Error_1:
				IF(NOT Reset) THEN
					DiagCode := TO_WORD(SF_EDM_State#Init);
				END_IF;
			SF_EDM_State#Init_Error:
				IF(NOT Reset) THEN
					DiagCode := TO_WORD(SF_EDM_State#Init);
				END_IF;
			SF_EDM_State#Output_Disable:
				MonitoringTimer_OutputDisable();
				//NOTE: priorities are definied exactly in this way, because otherwise some states would be unreachable!
				IF(IS(S_OutControl) AND NOT EDM1 AND NOT EDM2) THEN
					DiagCode := TO_WORD(SF_EDM_State#EDM_Error_13);
				ELSIF(IS(S_OutControl) AND NOT EDM1) THEN
					DiagCode := TO_WORD(SF_EDM_State#EDM_Error_11);
				ELSIF(IS(S_OutControl) AND NOT EDM2) THEN
					DiagCode := TO_WORD(SF_EDM_State#EDM_Error_12);
				ELSIF(MonitoringTimer_OutputDisable.Q AND NOT EDM1 AND NOT EDM2) THEN
					DiagCode := TO_WORD(SF_EDM_State#EDM_Error_23);
				ELSIF(MonitoringTimer_OutputDisable.Q AND NOT EDM1) THEN
					DiagCode := TO_WORD(SF_EDM_State#EDM_Error_21);
				ELSIF(MonitoringTimer_OutputDisable.Q AND NOT EDM2) THEN
					DiagCode := TO_WORD(SF_EDM_State#EDM_Error_22);
				ELSIF(IS(S_OutControl)) THEN
					DiagCode := TO_WORD(SF_EDM_State#Output_Enable);
				END_IF;
			SF_EDM_State#EDM_Error_11:
				IF((Reset AND NOT R_Trig_Reset.Q AND EDM1 AND EDM2) OR (R_Trig_Reset.Q AND R_Trig_EDM1.Q)) THEN
					DiagCode := TO_WORD(SF_EDM_State#Reset_Error_21);
				ELSIF(R_Trig_Reset.Q AND EDM1 AND EDM2) THEN
					DiagCode := TO_WORD(SF_EDM_State#Output_Disable);
				END_IF;
			SF_EDM_State#EDM_Error_12:
				IF((Reset AND NOT R_Trig_Reset.Q AND EDM1 AND EDM2) OR (R_Trig_Reset.Q AND R_Trig_EDM2.Q)) THEN
					DiagCode := TO_WORD(SF_EDM_State#Reset_Error_22);
				ELSIF(R_Trig_Reset.Q AND EDM1 AND EDM2) THEN
					DiagCode := TO_WORD(SF_EDM_State#Output_Disable);
				END_IF;
			SF_EDM_State#EDM_Error_13:
				IF((Reset AND NOT R_Trig_Reset.Q AND EDM1 AND EDM2) OR (R_Trig_Reset.Q AND R_Trig_EDM1.Q AND R_Trig_EDM2.Q)) THEN
					DiagCode := TO_WORD(SF_EDM_State#Reset_Error_23);
				ELSIF(R_Trig_Reset.Q AND EDM1 AND EDM2) THEN
					DiagCode := TO_WORD(SF_EDM_State#Output_Disable);
				END_IF;
			SF_EDM_State#Reset_Error_21:
				IF(NOT Reset) THEN
					DiagCode := TO_WORD(SF_EDM_State#EDM_Error_11);
				END_IF;
			SF_EDM_State#Reset_Error_22:
				IF(NOT Reset) THEN
					DiagCode := TO_WORD(SF_EDM_State#EDM_Error_12);
				END_IF;
			SF_EDM_State#Reset_Error_23:
				IF(NOT Reset) THEN
					DiagCode := TO_WORD(SF_EDM_State#EDM_Error_13);
				END_IF;
			SF_EDM_State#EDM_Error_21:
				IF((Reset AND NOT R_Trig_Reset.Q AND EDM1 AND EDM2) OR (R_Trig_Reset.Q AND R_Trig_EDM1.Q)) THEN
					DiagCode := TO_WORD(SF_EDM_State#Reset_Error_31);
				ELSIF(R_Trig_Reset.Q AND EDM1 AND EDM2) THEN
					DiagCode := TO_WORD(SF_EDM_State#Output_Disable);
				END_IF;
			SF_EDM_State#EDM_Error_22:
				IF((Reset AND NOT R_Trig_Reset.Q AND EDM1 AND EDM2) OR (R_Trig_Reset.Q AND R_Trig_EDM2.Q)) THEN
					DiagCode := TO_WORD(SF_EDM_State#Reset_Error_32);
				ELSIF(R_Trig_Reset.Q AND EDM1 AND EDM2) THEN
					DiagCode := TO_WORD(SF_EDM_State#Output_Disable);
				END_IF;
			SF_EDM_State#EDM_Error_23:
				IF((Reset AND NOT R_Trig_Reset.Q AND EDM1 AND EDM2) OR (R_Trig_Reset.Q AND R_Trig_EDM1.Q AND R_Trig_EDM2.Q)) THEN
					DiagCode := TO_WORD(SF_EDM_State#Reset_Error_33);
				ELSIF(R_Trig_Reset.Q AND EDM1 AND EDM2) THEN
					DiagCode := TO_WORD(SF_EDM_State#Output_Disable);
				END_IF;
			SF_EDM_State#Reset_Error_31:
				IF(NOT Reset) THEN
					DiagCode := TO_WORD(SF_EDM_State#EDM_Error_21);
				END_IF;
			SF_EDM_State#Reset_Error_32:
				IF(NOT Reset) THEN
					DiagCode := TO_WORD(SF_EDM_State#EDM_Error_22);
				END_IF;
			SF_EDM_State#Reset_Error_33:
				IF(NOT Reset) THEN
					DiagCode := TO_WORD(SF_EDM_State#EDM_Error_23);
				END_IF;
			SF_EDM_State#Output_Enable:
				MonitoringTimer_OutputEnable();
				//NOTE: priorities are definied exactly in this way, because otherwise some states would be unreachable!
				IF(MonitoringTimer_OutputEnable.Q AND EDM1 AND EDM2) THEN
					DiagCode := TO_WORD(SF_EDM_State#EDM_Error_33);
				ELSIF(MonitoringTimer_OutputEnable.Q AND EDM1) THEN
					DiagCode := TO_WORD(SF_EDM_State#EDM_Error_31);
				ELSIF(MonitoringTimer_OutputEnable.Q AND EDM2) THEN
					DiagCode := TO_WORD(SF_EDM_State#EDM_Error_32);
				ELSIF(IS_NOT(S_OutControl)) THEN
					DiagCode := TO_WORD(SF_EDM_State#Output_Disable);
				END_IF;
			SF_EDM_State#EDM_Error_31:
				IF(Reset AND NOT R_Trig_Reset.Q) THEN
					DiagCode := TO_WORD(SF_EDM_State#Reset_Error_41);
				ELSIF(R_Trig_Reset.Q AND NOT (R_Trig_EDM1.Q OR R_Trig_EDM2.Q)) THEN
					DiagCode := TO_WORD(SF_EDM_State#Output_Disable);
				END_IF;
			SF_EDM_State#EDM_Error_32:
				IF(Reset AND NOT R_Trig_Reset.Q) THEN
					DiagCode := TO_WORD(SF_EDM_State#Reset_Error_42);
				ELSIF(R_Trig_Reset.Q AND NOT (R_Trig_EDM1.Q OR R_Trig_EDM2.Q)) THEN
					DiagCode := TO_WORD(SF_EDM_State#Output_Disable);
				END_IF;
			SF_EDM_State#EDM_Error_33:
				IF(Reset AND NOT R_Trig_Reset.Q) THEN
					DiagCode := TO_WORD(SF_EDM_State#Reset_Error_43);
				ELSIF(R_Trig_Reset.Q AND NOT (R_Trig_EDM1.Q OR R_Trig_EDM2.Q)) THEN
					DiagCode := TO_WORD(SF_EDM_State#Output_Disable);
				END_IF;
			SF_EDM_State#Reset_Error_41:
				IF(NOT Reset) THEN
					DiagCode := TO_WORD(SF_EDM_State#EDM_Error_31);
				END_IF;
			SF_EDM_State#Reset_Error_42:
				IF(NOT Reset) THEN
					DiagCode := TO_WORD(SF_EDM_State#EDM_Error_32);
				END_IF;
			SF_EDM_State#Reset_Error_43:
				IF(NOT Reset) THEN
					DiagCode := TO_WORD(SF_EDM_State#EDM_Error_33);
				END_IF;
		END_CASE;
	END_IF;

	CASE TO_UINT(DiagCode) OF
		SF_EDM_State#Idle:
			MonitoringTimer_OutputDisable(IN := FALSE);
			MonitoringTimer_OutputEnable(IN := FALSE);
			Ready := FALSE;
			S_EDM_Out := SAFEBOOL_Constant#SAFEFALSE;
			SafetyDemand := FALSE;
			ResetRequest := FALSE;
			Error := FALSE;
		SF_EDM_State#Init:
			MonitoringTimer_OutputDisable(IN := FALSE);
			MonitoringTimer_OutputEnable(IN := FALSE);
			Ready := TRUE;
			S_EDM_Out := SAFEBOOL_Constant#SAFEFALSE;
			SafetyDemand := FALSE;
			ResetRequest := TRUE;
			Error := FALSE;
		SF_EDM_State#Output_Disable:
			MonitoringTimer_OutputDisable(IN := TRUE, PT := MonitoringTime);
			MonitoringTimer_OutputEnable(IN := FALSE);
			Ready := TRUE;
			S_EDM_Out := SAFEBOOL_Constant#SAFEFALSE;
			SafetyDemand := TRUE;
			ResetRequest := FALSE;
			Error := FALSE;
		SF_EDM_State#Output_Enable:
			MonitoringTimer_OutputEnable(IN := TRUE, PT := MonitoringTime);
			MonitoringTimer_OutputDisable(IN := FALSE);
			Ready := TRUE;
			S_EDM_Out := SAFEBOOL_Constant#SAFETRUE;
			SafetyDemand := FALSE;
			ResetRequest := FALSE;
			Error := FALSE;
		SF_EDM_State#Reset_Error_1,
		SF_EDM_State#Reset_Error_21,
		SF_EDM_State#Reset_Error_22,
		SF_EDM_State#Reset_Error_23,
		SF_EDM_State#Reset_Error_31,
		SF_EDM_State#Reset_Error_32,
		SF_EDM_State#Reset_Error_33,
		SF_EDM_State#Reset_Error_41,
		SF_EDM_State#Reset_Error_42,
		SF_EDM_State#Reset_Error_43,
		SF_EDM_State#EDM_Error_13,
		SF_EDM_State#Init_Error:
			MonitoringTimer_OutputDisable(IN := FALSE);
			MonitoringTimer_OutputEnable(IN := FALSE);
			Ready := TRUE;
			S_EDM_Out := SAFEBOOL_Constant#SAFEFALSE;
			SafetyDemand := FALSE;
			ResetRequest := FALSE;
			Error := TRUE;
		SF_EDM_State#EDM_Error_11,
		SF_EDM_State#EDM_Error_12,
		SF_EDM_State#EDM_Error_21,
		SF_EDM_State#EDM_Error_22,
		SF_EDM_State#EDM_Error_23:
			MonitoringTimer_OutputDisable(IN := FALSE);
			MonitoringTimer_OutputEnable(IN := FALSE);
			Ready := TRUE;
			S_EDM_Out := SAFEBOOL_Constant#SAFEFALSE;
			SafetyDemand := FALSE;
			ResetRequest := FALSE;
			Error := TRUE;
		SF_EDM_State#EDM_Error_31,
		SF_EDM_State#EDM_Error_32,
		SF_EDM_State#EDM_Error_33:
			MonitoringTimer_OutputDisable(IN := FALSE);
			MonitoringTimer_OutputEnable(IN := FALSE);
			Ready := TRUE;
			S_EDM_Out := SAFEBOOL_Constant#SAFEFALSE;
			SafetyDemand := FALSE;
			ResetRequest := TRUE;
			Error := TRUE;
	END_CASE;

	ENO := ENO AND CheckSAFEBOOL(S_OutControl);

END_FUNCTION_BLOCK

END_NAMESPACE
END_NAMESPACE

(* ---- SF_EmergencyStop.iecst ---- *)
USING logicals.web.standard.safe;

NAMESPACE logicals.web.standard.safe
NAMESPACE plcopen

/*
 * This function block is a safety-related function block for monitoring an emergency stop button.
 * This FB can be used for emergency switch off functionality (stop category 0),
 * or - with additional peripheral support - as emergency stop (stop category 1 or 2)
 */
FUNCTION_BLOCK SF_EmergencyStop
	{ altName:="SF_EmergencyStop"; bgColor:="Gold"; width:=380; }
	VAR_INPUT
		/* See Section 5.1.1 General Input Parameters */
		Activate : BOOL := FALSE;
		/* Safety demand input.
		 * Variable.
		 * FALSE: Demand for safety-related response (e.g., emergency stop button is engaged).
		 * TRUE: No demand for safety-related response (e.g., emergen-cy stop button not engaged).
		 */
		S_EStopIn : SAFEBOOL := SAFEBOOL_Constant#SAFEFALSE;
		/* See Section 5.1.1 General Input Parameters */
		S_StartReset : SAFEBOOL := SAFEBOOL_Constant#SAFEFALSE;
		/* See Section 5.1.1 General Input Parameters */
		S_AutoReset : SAFEBOOL := SAFEBOOL_Constant#SAFEFALSE;
		/* See Section 5.1.1 General Input Parameters */
		Reset : BOOL := FALSE;
	END_VAR
	VAR_OUTPUT
		/* See Section 5.1.2 General Output Parameters */
		Ready : BOOL := FALSE;
		/* Output for the safety-related response.
		 * FALSE: Safety output disabled. Demand for safety-related response (e.g., emergency stop button engaged, reset required or internal errors active)
		 * TRUE: Safety output enabled. No demand for safety-related response (e.g., emergency stop button not engaged, no internal errors active).
		 */
		S_EStopOut : SAFEBOOL := SAFEBOOL_Constant#SAFEFALSE;
		/* Optional. See 5.1.2 General Output Parameters */
		SafetyDemand : BOOL := FALSE;
		/* Optional. See 5.1.2 General Output Parameters */
		ResetRequest : BOOL := FALSE;
		/* See Section 5.1.2 General Output Parameters */
		Error : BOOL := FALSE;
		/* See Section 5.1.2 General Output Parameters */
		DiagCode : WORD := 16#0000;
	END_VAR
	VAR
		GenericSafetyDemand : SFB_GenericSafetyDemand;
	END_VAR

	GenericSafetyDemand(
		Activate := Activate,
		S_SafetyDemandIn := S_EStopIn,
		S_StartReset := S_StartReset,
		S_AutoReset := S_AutoReset,
		Reset := Reset,
		Ready => Ready,
		S_SafetyDemandOut => S_EStopOut,
		SafetyDemand => SafetyDemand,
		ResetRequest => ResetRequest,
		Error => Error,
		DiagCode => DiagCode,
		ENO => ENO
	);

END_FUNCTION_BLOCK

END_NAMESPACE
END_NAMESPACE

(* ---- SF_EnableSwitch.iecst ---- *)
USING logicals.web.standard.safe;

NAMESPACE logicals.web.standard.safe
NAMESPACE plcopen

TYPE
	SF_EnableSwitch_State : UINT(
	/* Static Reset signal detected in state C020. */
	Reset_Error_1 := 16#C001,
	/* Static Reset signal detected in state C040. */
	Reset_Error_2 := 16#C011,
	/* Enable switch not in position 1 during activation of S_SafetyActive. */
	Operation_Error_1 := 16#C010,
	/* Enable switch in position 1 after C010. */
	Operation_Error_2 := 16#C020,
	/* Enable switch in position 2 after position 3. */
	Operation_Error_3 := 16#C030,
	/* Enable switch not in position 2 after C030. */
	Operation_Error_4 := 16#C040,
	/* The function block is not active (initial state). */
	Idle := 16#0000,
	/* Safe operation mode is not active. */
	Basic_Operation_Mode := 16#8002,
	/* Safe operation mode is active. */
	Safe_Operation_Mode := 16#8004,
	/* Safe operation mode is active and the enable switch is in position 1. */
	Position_1 := 16#8802,
	/* Safe operation mode is active and the enable switch is in position 3. */
	Position_3 := 16#8804,
	/* Safe operation mode is active and the enable switch is in position 2. */
	Position_2 := 16#8000
	);
END_TYPE

/* The SF_EnableSwitch FB evaluates the signals of an enable switch with three positions. */

FUNCTION_BLOCK SF_EnableSwitch
	{ altName := "SF_EnableSwitch"; bgColor := "Gold"; width := 440;}
	VAR_INPUT
		/* See Section 5.1.1 General Input Parameters */
		Activate : BOOL := FALSE;
		/* Variable or constant.
		 * Confirmation of the safe mode (limitation of the speed or the power of motion, limitation of the range of mo-tion).
		 * FALSE: Safe mode is not active.
		 * TRUE: Safe mode is active.
		 */
		S_SafetyActive : SAFEBOOL := SAFEBOOL_Constant#SAFEFALSE;
		/* Variable.
		 * Signal of contacts E1 and E2 of the connected enable switch.
		 * FALSE: Connected switches are open.
		 * TRUE: Connected switches are closed.
		 */
		S_EnableSwitchCh1 : SAFEBOOL := SAFEBOOL_Constant#SAFEFALSE;
		/* Variable.
		 * Signal of contacts E3 and E4 of the connected enable switch.
		 * FALSE: Connected switches are open.
		 * TRUE: Connected switches are closed.
		 */
		S_EnableSwitchCh2 : SAFEBOOL := SAFEBOOL_Constant#SAFEFALSE;
		/* See Section 5.1.1 General Input Parameters */
		S_AutoReset : SAFEBOOL := SAFEBOOL_Constant#SAFEFALSE;
		/* See Section 5.1.1 General Input Parameters */
		Reset : BOOL := FALSE;
	END_VAR
	VAR_OUTPUT
		/* See 5.1.2 General Output Parameters */
		Ready : BOOL := FALSE;
		/* Safety related output: Indicates suspension of guard.
		 * FALSE: Disable suspension of safeguarding.
		 * TRUE: Enable suspension of safeguarding.
		 */
		S_EnableSwitchOut : SAFEBOOL := SAFEBOOL_Constant#SAFEFALSE;
		/* See 5.1.2 General Output Parameters */
		SafetyDemand : BOOL := FALSE;
		/* See 5.1.2 General Output Parameters */
		ResetRequest : BOOL := FALSE;
		/* See Section 5.1.2 General Output Parameters */
		Error : BOOL := FALSE;
		/* See Section 5.1.2 General Output Parameters */
		DiagCode : WORD := 16#0000;
	END_VAR
	VAR
		R_Trig_Reset : R_TRIG;
	END_VAR

	R_Trig_Reset(Reset);

	IF(NOT Activate) THEN
		DiagCode := TO_WORD(SF_EnableSwitch_State#Idle);
	ELSE
		CASE TO_UINT(DiagCode) OF
			SF_EnableSwitch_State#Idle:
				/* IF(Activate) THEN - Activate is always true here */
					DiagCode := TO_WORD(SF_EnableSwitch_State#Basic_Operation_Mode);
			SF_EnableSwitch_State#Basic_Operation_Mode:
				IF(IS(S_SafetyActive)) THEN
					DiagCode := TO_WORD(SF_EnableSwitch_State#Safe_Operation_Mode);
				END_IF;
			SF_EnableSwitch_State#Safe_Operation_Mode:
				IF(IS_NOT(S_SafetyActive)) THEN
					DiagCode := TO_WORD(SF_EnableSwitch_State#Basic_Operation_Mode);
				ELSIF(NOT(IS_NOT(S_EnableSwitchCh1) AND IS(S_EnableSwitchCh2))) THEN
					DiagCode := TO_WORD(SF_EnableSwitch_State#Operation_Error_1);
				/* ELSIF(IS_NOT(S_EnableSwitchCh1) AND IS(S_EnableSwitchCh2)) THEN */
				ELSE
					DiagCode := TO_WORD(SF_EnableSwitch_State#Position_1);
				END_IF;
			SF_EnableSwitch_State#Operation_Error_1:
				IF(IS_NOT(S_SafetyActive)) THEN
					DiagCode := TO_WORD(SF_EnableSwitch_State#Basic_Operation_Mode);
				ELSIF(IS_NOT(S_EnableSwitchCh1) AND IS(S_EnableSwitchCh2)) THEN
					DiagCode := TO_WORD(SF_EnableSwitch_State#Operation_Error_2);
				END_IF;
			SF_EnableSwitch_State#Operation_Error_2:
				IF(IS_NOT(S_SafetyActive)) THEN
					DiagCode := TO_WORD(SF_EnableSwitch_State#Basic_Operation_Mode);
				ELSIF(NOT(IS_NOT(S_EnableSwitchCh1) AND IS(S_EnableSwitchCh2))) THEN
					DiagCode := TO_WORD(SF_EnableSwitch_State#Operation_Error_1);
				ELSIF(Reset AND NOT R_Trig_Reset.Q AND IS_NOT(S_AutoReset)) THEN
					DiagCode := TO_WORD(SF_EnableSwitch_State#Reset_Error_1);
				ELSIF(R_Trig_Reset.Q OR IS(S_AutoReset)) THEN
					DiagCode := TO_WORD(SF_EnableSwitch_State#Position_1);
				END_IF;
			SF_EnableSwitch_State#Reset_Error_1:
				IF(IS_NOT(S_SafetyActive)) THEN
					DiagCode := TO_WORD(SF_EnableSwitch_State#Basic_Operation_Mode);
				ELSIF(NOT Reset) THEN
					DiagCode := TO_WORD(SF_EnableSwitch_State#Operation_Error_2);
				END_IF;
			SF_EnableSwitch_State#Position_1:
				IF(IS_NOT(S_SafetyActive)) THEN
					DiagCode := TO_WORD(SF_EnableSwitch_State#Basic_Operation_Mode);
				ELSIF(IS(S_EnableSwitchCh1) AND IS(S_EnableSwitchCh2)) THEN
					DiagCode := TO_WORD(SF_EnableSwitch_State#Position_2);
				ELSIF(NOT (IS(S_EnableSwitchCh1) OR IS(S_EnableSwitchCh2))) THEN
					DiagCode := TO_WORD(SF_EnableSwitch_State#Position_3);
				END_IF;
			SF_EnableSwitch_State#Position_3:
				IF(IS_NOT(S_SafetyActive)) THEN
					DiagCode := TO_WORD(SF_EnableSwitch_State#Basic_Operation_Mode);
				ELSIF(IS(S_EnableSwitchCh1) AND IS(S_EnableSwitchCh2)) THEN
					DiagCode := TO_WORD(SF_EnableSwitch_State#Operation_Error_3);
				ELSIF(NOT IS(S_EnableSwitchCh1) AND IS(S_EnableSwitchCh2)) THEN
					DiagCode := TO_WORD(SF_EnableSwitch_State#Position_1);
				END_IF;
			SF_EnableSwitch_State#Operation_Error_4:
				IF(IS_NOT(S_SafetyActive)) THEN
					DiagCode := TO_WORD(SF_EnableSwitch_State#Basic_Operation_Mode);
				ELSIF(IS(S_EnableSwitchCh1) AND IS(S_EnableSwitchCh2)) THEN
					DiagCode := TO_WORD(SF_EnableSwitch_State#Operation_Error_3);
				ELSIF(Reset AND NOT R_Trig_Reset.Q AND IS_NOT(S_AutoReset)) THEN
					DiagCode := TO_WORD(SF_EnableSwitch_State#Reset_Error_2);
				ELSIF(R_Trig_Reset.Q OR IS(S_AutoReset)) THEN
					DiagCode := TO_WORD(SF_EnableSwitch_State#Position_3);
				END_IF;
			SF_EnableSwitch_State#Operation_Error_3:
				IF(IS_NOT(S_SafetyActive)) THEN
					DiagCode := TO_WORD(SF_EnableSwitch_State#Basic_Operation_Mode);
				ELSIF(NOT(IS(S_EnableSwitchCh1) AND IS(S_EnableSwitchCh2))) THEN
					DiagCode := TO_WORD(SF_EnableSwitch_State#Operation_Error_4);
				END_IF;
			SF_EnableSwitch_State#Reset_Error_2:
				IF(IS_NOT(S_SafetyActive)) THEN
					DiagCode := TO_WORD(SF_EnableSwitch_State#Basic_Operation_Mode);
				ELSIF(NOT Reset) THEN
					DiagCode := TO_WORD(SF_EnableSwitch_State#Operation_Error_4);
				END_IF;
			SF_EnableSwitch_State#Position_2:
				IF(IS_NOT(S_SafetyActive)) THEN
					DiagCode := TO_WORD(SF_EnableSwitch_State#Basic_Operation_Mode);
				ELSIF(NOT(IS(S_EnableSwitchCh1) OR IS(S_EnableSwitchCh2))) THEN
					DiagCode := TO_WORD(SF_EnableSwitch_State#Position_3);
				ELSIF(IS_NOT(S_EnableSwitchCh1) AND IS(S_EnableSwitchCh2)) THEN
					DiagCode := TO_WORD(SF_EnableSwitch_State#Position_1);
				END_IF;
			ELSE
				ENO := FALSE;
		END_CASE;
	END_IF;

		CASE TO_UINT(DiagCode) OF
			SF_EnableSwitch_State#Reset_Error_1,
			SF_EnableSwitch_State#Reset_Error_2,
			SF_EnableSwitch_State#Operation_Error_1,
			SF_EnableSwitch_State#Operation_Error_3:
				Ready := TRUE;
				S_EnableSwitchOut := SAFEBOOL_Constant#SAFEFALSE;
				SafetyDemand := FALSE;
				ResetRequest := FALSE;
				Error := TRUE;
			SF_EnableSwitch_State#Operation_Error_2,
			SF_EnableSwitch_State#Operation_Error_4:
				Ready := TRUE;
				S_EnableSwitchOut := SAFEBOOL_Constant#SAFEFALSE;
				SafetyDemand := FALSE;
				ResetRequest := TRUE;
				Error := TRUE;
			SF_EnableSwitch_State#Idle:
				Ready := FALSE;
				S_EnableSwitchOut := SAFEBOOL_Constant#SAFEFALSE;
				SafetyDemand := FALSE;
				ResetRequest := FALSE;
				Error := FALSE;
			SF_EnableSwitch_State#Basic_Operation_Mode,
			SF_EnableSwitch_State#Safe_Operation_Mode:
				Ready := TRUE;
				S_EnableSwitchOut := SAFEBOOL_Constant#SAFEFALSE;
				SafetyDemand := FALSE;
				ResetRequest := FALSE;
				Error := FALSE;
			SF_EnableSwitch_State#Position_1,
			SF_EnableSwitch_State#Position_3:
				Ready := TRUE;
				S_EnableSwitchOut := SAFEBOOL_Constant#SAFEFALSE;
				SafetyDemand := TRUE;
				ResetRequest := FALSE;
				Error := FALSE;
			SF_EnableSwitch_State#Position_2:
				Ready := TRUE;
				S_EnableSwitchOut := SAFEBOOL_Constant#SAFETRUE;
				SafetyDemand := FALSE;
				ResetRequest := FALSE;
				Error := FALSE;
			ELSE
				ENO := FALSE;
		END_CASE;

		ENO := ENO AND CheckSAFEBOOL(S_SafetyActive) AND CheckSAFEBOOL(S_EnableSwitchCh1) AND CheckSAFEBOOL(S_EnableSwitchCh2) AND CheckSAFEBOOL(S_AutoReset);

END_FUNCTION_BLOCK

END_NAMESPACE
END_NAMESPACE

(* ---- SF_EnableSwitch_2.iecst ---- *)
USING logicals.web.standard.safe;

NAMESPACE logicals.web.standard.safe
NAMESPACE plcopen

TYPE
	SF_EnableSwitch_2_State : UINT(
	/* Static Reset signal detected in state Cx10. */
	Reset_Error_1 := 16#C001,
	/* Enable switch in position 2 during activation of S_SafetyActive. */
	Operation_Error_1_Position_2 := 16#C010,
	/* Enable switch in position 1 or 3 during activation of S_SafetyActive. */
	Operation_Error_1_Position_1_Or_3 := 16#C410,
	/* The function block is not active (initial state). */
	Idle := 16#0000,
	/* Safe operation mode is not active. */
	Basic_Operation_Mode := 16#8002,
	/* Safe operation mode is active. */
	Safe_Operation_Mode := 16#8004,
	/* Safe operation mode is active and the enable switch is in position 1 or 3. */
	Position_1_Or_3 := 16#8802,
	/* Safe operation mode is active and the enable switch is in position 2. */
	Position_2 := 16#8000
	);
END_TYPE

/**
 * The SF_EnableSwitch_2 evaluates the signals of an enable switch with two or three positions.
 */
FUNCTION_BLOCK SF_EnableSwitch_2
	{ altName:="SF_EnableSwitch_2"; bgColor:="Gold"; width:=380;}
	VAR_INPUT
		/* See 5.1.1 General Input Parameters */
		Activate : BOOL := FALSE;
		/* Variable or constant.
		 * Confirmation of the safe mode (limitation of the speed or the power of motion, limitation of the range of mo-tion).
		 * FALSE: Safe mode is not active.
		 * TRUE: Safe mode is active. */
		S_SafetyActive : SAFEBOOL := SAFEBOOL_Constant#SAFEFALSE;
		/* Variable.
		 * Signal of connected enable switch. The evaluation of the signals (discrepancy) will be done within the IO unit or the FB_Equivalent
		 * FALSE: Not Enabled.
		 * TRUE: Enabled. */
		S_EnableIn : SAFEBOOL := SAFEBOOL_Constant#SAFEFALSE;
		/* See 5.1.1 General Input Parameters */
		Reset : BOOL := FALSE;
	END_VAR

	VAR_OUTPUT
		/* See 5.1.2 General Output Parameters */
		Ready : BOOL := FALSE;
		/* Safety related output: Indicates suspension of guard.
		 * FALSE: Disable suspension of safeguarding.
		 * TRUE: Enable suspension of safeguarding. */
		S_EnableSwitchOut : SAFEBOOL := SAFEBOOL_Constant#SAFEFALSE;
		/* See 5.1.2 General Output Parameters */
		SafetyDemand : BOOL := FALSE;
		/* See 5.1.2 General Output Parameters */
		ResetRequest : BOOL := FALSE;
		/* See 5.1.2 General Output Parameters */
		Error : BOOL := FALSE;
		/* See 5.1.2 General Output Parameters */
		DiagCode : WORD := 16#0000;
	END_VAR

	VAR
		R_Trig_Reset : R_TRIG;
	END_VAR

	R_Trig_Reset(Reset);

	IF(NOT Activate) THEN
		DiagCode := TO_WORD(SF_EnableSwitch_2_State#Idle);
	ELSE
		CASE TO_UINT(DiagCode) OF
			SF_EnableSwitch_2_State#Idle:
				/* IF(Activate) THEN - Active is always TRUE here */
					DiagCode := TO_WORD(SF_EnableSwitch_2_State#Basic_Operation_Mode);
			SF_EnableSwitch_2_State#Basic_Operation_Mode:
				IF(IS(S_SafetyActive)) THEN
					DiagCode := TO_WORD(SF_EnableSwitch_2_State#Safe_Operation_Mode);
				END_IF;
			SF_EnableSwitch_2_State#Safe_Operation_Mode:
				IF(IS_NOT(S_SafetyActive)) THEN
					DiagCode := TO_WORD(SF_EnableSwitch_2_State#Basic_Operation_Mode);
				ELSIF(IS(S_EnableIn)) THEN
					DiagCode := TO_WORD(SF_EnableSwitch_2_State#Operation_Error_1_Position_2);
				/* ELSIF(IS_NOT(S_EnableIn)) THEN - S_EnableIn can only be FALSE here */
				ELSE
					DiagCode := TO_WORD(SF_EnableSwitch_2_State#Position_1_Or_3);
				END_IF;
			SF_EnableSwitch_2_State#Operation_Error_1_Position_2,
			SF_EnableSwitch_2_State#Operation_Error_1_Position_1_Or_3:
				IF(IS_NOT(S_SafetyActive)) THEN
					DiagCode := TO_WORD(SF_EnableSwitch_2_State#Basic_Operation_Mode);
				ELSIF(Reset AND NOT R_Trig_Reset.Q) THEN
					DiagCode := TO_WORD(SF_EnableSwitch_2_State#Reset_Error_1);
				ELSIF(IS_NOT(S_EnableIn) AND R_Trig_Reset.Q) THEN
					DiagCode := TO_WORD(SF_EnableSwitch_2_State#Position_1_Or_3);
				END_IF;
			SF_EnableSwitch_2_State#Reset_Error_1:
				IF(IS_NOT(S_SafetyActive)) THEN
					DiagCode := TO_WORD(SF_EnableSwitch_2_State#Basic_Operation_Mode);
				ELSIF(NOT Reset) THEN
					IF(IS(S_EnableIn)) THEN
						DiagCode := TO_WORD(SF_EnableSwitch_2_State#Operation_Error_1_Position_2);
					ELSE
						DiagCode := TO_WORD(SF_EnableSwitch_2_State#Operation_Error_1_Position_1_Or_3);
					END_IF;
				END_IF;
			SF_EnableSwitch_2_State#Position_1_Or_3:
				IF(IS_NOT(S_SafetyActive)) THEN
					DiagCode := TO_WORD(SF_EnableSwitch_2_State#Basic_Operation_Mode);
				ELSIF(IS(S_EnableIn)) THEN
					DiagCode := TO_WORD(SF_EnableSwitch_2_State#Position_2);
				END_IF;
			SF_EnableSwitch_2_State#Position_2:
				IF(IS_NOT(S_SafetyActive)) THEN
					DiagCode := TO_WORD(SF_EnableSwitch_2_State#Basic_Operation_Mode);
				ELSIF(IS_NOT(S_EnableIn)) THEN
					DiagCode := TO_WORD(SF_EnableSwitch_2_State#Position_1_Or_3);
				END_IF;
			ELSE
				ENO := FALSE;
		END_CASE;
	END_IF;

	CASE TO_UINT(DiagCode) OF
		SF_EnableSwitch_2_State#Idle:
			Ready := FALSE;
			S_EnableSwitchOut := SAFEBOOL_Constant#SAFEFALSE;
			SafetyDemand := FALSE;
			ResetRequest := FALSE;
			Error := FALSE;
		SF_EnableSwitch_2_State#Basic_Operation_Mode,
		SF_EnableSwitch_2_State#Safe_Operation_Mode:
			Ready := TRUE;
			S_EnableSwitchOut := SAFEBOOL_Constant#SAFEFALSE;
			SafetyDemand := FALSE;
			ResetRequest := FALSE;
			Error := FALSE;
		SF_EnableSwitch_2_State#Position_1_Or_3:
			Ready := TRUE;
			S_EnableSwitchOut := SAFEBOOL_Constant#SAFEFALSE;
			SafetyDemand := TRUE;
			ResetRequest := FALSE;
			Error := FALSE;
		SF_EnableSwitch_2_State#Position_2:
			Ready := TRUE;
			S_EnableSwitchOut := SAFEBOOL_Constant#SAFETRUE;
			SafetyDemand := FALSE;
			ResetRequest := FALSE;
			Error := FALSE;
		SF_EnableSwitch_2_State#Reset_Error_1,
		SF_EnableSwitch_2_State#Operation_Error_1_Position_2:
			Ready := TRUE;
			S_EnableSwitchOut := SAFEBOOL_Constant#SAFEFALSE;
			SafetyDemand := FALSE;
			ResetRequest := FALSE;
			Error := TRUE;
		SF_EnableSwitch_2_State#Operation_Error_1_Position_1_Or_3:
			Ready := TRUE;
			S_EnableSwitchOut := SAFEBOOL_Constant#SAFEFALSE;
			SafetyDemand := FALSE;
			ResetRequest := TRUE;
			Error := TRUE;
		ELSE
			ENO := FALSE;
	END_CASE;

	ENO := ENO AND CheckSAFEBOOL(S_SafetyActive) AND CheckSAFEBOOL(S_EnableIn);

END_FUNCTION_BLOCK

END_NAMESPACE
END_NAMESPACE

(* ---- SF_Equivalent.iecst ---- *)
USING logicals.web.standard.safe;

NAMESPACE logicals.web.standard.safe
NAMESPACE plcopen

TYPE
	SF_Equivalent_State : UINT(
	/* Discrepancy time elapsed in state 8802. */
	Error_1 := 16#C010,
	/* Discrepancy time elapsed in state 8804. */
	Error_2 := 16#C020,
	/* Discrepancy time elapsed in state 8806. */
	Error_3 := 16#C030,
	/* The function block is not active (initial state). */
	Idle := 16#0000,
	/* An activation has been detected by the FB and the FB is now activated. */
	Init := 16#8801,
	/* Output Enabled. The inputs switched to TRUE in equivalent mode. */
	Safety_Output_Enabled := 16#8000,
	/* Channel A has been switched to TRUE - waiting for Channel B; discrepancy timer started. */
	Wait_for_Channel_B := 16#8802,
	/* Channel B has been switched to TRUE - waiting for Channel A; discrepancy timer started. */
	Wait_for_Channel_A := 16#8804,
	/* One channel has been switched to FALSE; waiting for the second channel to be switched to FALSE, discrepancy timer started. */
	From_Active_Wait := 16#8806
	);
END_TYPE

/*
 * This function block converts two equivalent SAFEBOOL inputs (both NO or NC) to one SAFEBOOL output, including discrepancy time monitoring.
 * This FB should not be used stand-alone since it has no restart interlock.
 * It is required to connect the output to other safety related functionalities.
 */
FUNCTION_BLOCK SF_Equivalent
	{ altName := "SF_Equivalent"; bgColor := "Gold"; width := 380; }
	VAR_INPUT
		/* See Section 5.1.1 General Input Parameters */
		Activate : BOOL := FALSE;
		/* Variable. Input A for logical connection.
		 * FALSE: Contact A open
		 * TRUE: Contact A closed. */
		S_ChannelA : SAFEBOOL := SAFEBOOL_Constant#SAFEFALSE;
		/* Variable. Input B for logical connection.
		 * FALSE: Contact B open
		 * TRUE: Contact B closed. */
		S_ChannelB : SAFEBOOL := SAFEBOOL_Constant#SAFEFALSE;
		/* Constant. Maximum monitoring time for discrepancy status of both inputs. */
		DiscrepancyTime : TIME := T#0ms;
	END_VAR
	VAR_OUTPUT
		/* See Section 5.1.2 General Output Parameters */
		Ready : BOOL := FALSE;
		/* Safety related output
		 * FALSE: Minimum of one input signal = "FALSE" or status change outside of monitoring time.
		 * TRUE: Both input signals "active" and status change within monitoring time. */
		S_EquivalentOut : SAFEBOOL := SAFEBOOL_Constant#SAFEFALSE;
		/* Optional. See 5.1.2 General Output Parameters */
		SafetyDemand : BOOL := FALSE;
		/* See Section 5.1.2 General Output Parameters */
		Error : BOOL := FALSE;
		/* See Section 5.1.2 General Output Parameters */
		DiagCode : WORD := 16#0000;
	END_VAR
	VAR
		DiscrepancyTimer : TON;
	END_VAR

	IF(NOT Activate) THEN
		DiagCode := TO_WORD(SF_Equivalent_State#Idle);
	ELSE
		CASE TO_UINT(DiagCode) OF
			SF_Equivalent_State#Idle:
				/* IF(Activate) THEN - Active is always true here */
					DiagCode := TO_WORD(SF_Equivalent_State#Init);
			SF_Equivalent_State#Init:
				IF(IS(S_ChannelA) AND IS_NOT(S_ChannelB)) THEN
					DiagCode := TO_WORD(SF_Equivalent_State#Wait_for_Channel_B);
				ELSIF(IS(S_ChannelB) AND IS_NOT(S_ChannelA)) THEN
					DiagCode := TO_WORD(SF_Equivalent_State#Wait_for_Channel_A);
				ELSIF(IS(S_ChannelA) AND IS(S_ChannelB)) THEN
					DiagCode := TO_WORD(SF_Equivalent_State#Safety_Output_Enabled);
				END_IF;
			SF_Equivalent_State#Safety_Output_Enabled:
				IF(IS_NOT(S_ChannelA) AND IS_NOT(S_ChannelB)) THEN
					DiagCode := TO_WORD(SF_Equivalent_State#Init);
				ELSIF((S_ChannelA XOR S_ChannelB) <> 0) THEN
					DiagCode := TO_WORD(SF_Equivalent_State#From_Active_Wait);
				END_IF;
			SF_Equivalent_State#Wait_for_Channel_B:
				DiscrepancyTimer();
				IF(DiscrepancyTimer.Q) THEN
					DiagCode := TO_WORD(SF_Equivalent_State#Error_1);
				ELSIF(IS_NOT(S_ChannelA)) THEN
					DiagCode := TO_WORD(SF_Equivalent_State#Init);
				ELSIF(IS(S_ChannelB)) THEN
					DiagCode := TO_WORD(SF_Equivalent_State#Safety_Output_Enabled);
				END_IF;
			SF_Equivalent_State#Wait_for_Channel_A:
				DiscrepancyTimer();
				IF(DiscrepancyTimer.Q) THEN
					DiagCode := TO_WORD(SF_Equivalent_State#Error_2);
				ELSIF(IS_NOT(S_ChannelB)) THEN
					DiagCode := TO_WORD(SF_Equivalent_State#Init);
				ELSIF(IS(S_ChannelA)) THEN
					DiagCode := TO_WORD(SF_Equivalent_State#Safety_Output_Enabled);
				END_IF;
			SF_Equivalent_State#From_Active_Wait:
				DiscrepancyTimer();
				IF(DiscrepancyTimer.Q) THEN
					DiagCode := TO_WORD(SF_Equivalent_State#Error_3);
				ELSIF(IS_NOT(S_ChannelA) AND IS_NOT(S_ChannelB)) THEN
					DiagCode := TO_WORD(SF_Equivalent_State#Init);
				END_IF;
			SF_Equivalent_State#Error_1, SF_Equivalent_State#Error_2, SF_Equivalent_State#Error_3:
				IF(IS_NOT(S_ChannelA) AND IS_NOT(S_ChannelB)) THEN
					DiagCode := TO_WORD(SF_Equivalent_State#Init);
				END_IF;
			ELSE
				ENO := FALSE;
		END_CASE;
	END_IF;

	CASE TO_UINT(DiagCode) OF
		SF_Equivalent_State#Idle:
			DiscrepancyTimer(IN := FALSE);
			Ready := FALSE;
			S_EquivalentOut := SAFEBOOL_Constant#SAFEFALSE;
			SafetyDemand := FALSE;
			Error := FALSE;
		SF_Equivalent_State#Init:
			DiscrepancyTimer(IN := FALSE);
			Ready := TRUE;
			S_EquivalentOut := SAFEBOOL_Constant#SAFEFALSE;
			SafetyDemand := TRUE;
			Error := FALSE;
		SF_Equivalent_State#Safety_Output_Enabled:
			DiscrepancyTimer(IN := FALSE);
			Ready := TRUE;
			S_EquivalentOut := SAFEBOOL_Constant#SAFETRUE;
			SafetyDemand := FALSE;
			Error := FALSE;
		SF_Equivalent_State#Wait_for_Channel_B,SF_Equivalent_State#Wait_for_Channel_A,SF_Equivalent_State#From_Active_Wait:
			DiscrepancyTimer(IN := TRUE, PT := DiscrepancyTime);
			Ready := TRUE;
			S_EquivalentOut := SAFEBOOL_Constant#SAFEFALSE;
			SafetyDemand := TRUE;
			Error := FALSE;
		SF_Equivalent_State#Error_1,SF_Equivalent_State#Error_2,SF_Equivalent_State#Error_3:
			DiscrepancyTimer(IN := FALSE);
			Ready := TRUE;
			S_EquivalentOut := SAFEBOOL_Constant#SAFEFALSE;
			SafetyDemand := FALSE;
			Error := TRUE;
		ELSE
			ENO := FALSE;
	END_CASE;

	ENO := ENO AND CheckSAFEBOOL(S_ChannelA) AND CheckSAFEBOOL(S_ChannelB);

END_FUNCTION_BLOCK

END_NAMESPACE
END_NAMESPACE

(* ---- SF_ESPE.iecst ---- *)
USING logicals.web.standard.safe;

NAMESPACE logicals.web.standard.safe
NAMESPACE plcopen

/*
 * This function block is a safety-related function block for monitoring electro-sensitive protective equipment (ESPE).
 */
FUNCTION_BLOCK SF_ESPE
	{ altName:="SF_ESPE"; bgColor:="Gold"; width:=320; }
	VAR_INPUT
		/* See Section 5.1.1 General Input Parameters */
		Activate : BOOL := FALSE;
		/* Safety demand input.
		 * Variable.
		 * FALSE: ESPE actuated, demand for safety-related response.
		 * TRUE: ESPE not actuated, no demand for safety-related response.
		 * Safety control system must be able to detect a very short interruption of the sensor
		 * (which is specified in 61496-1: minimum 80 ms), when the ESPE is used in applications as a trip device
		 */
		S_ESPE_In : SAFEBOOL := SAFEBOOL_Constant#SAFEFALSE;
		/* See Section 5.1.1 General Input Parameters */
		S_StartReset : SAFEBOOL := SAFEBOOL_Constant#SAFEFALSE;
		/* See Section 5.1.1 General Input Parameters */
		S_AutoReset : SAFEBOOL := SAFEBOOL_Constant#SAFEFALSE;
		/* See Section 5.1.1 General Input Parameters */
		Reset : BOOL := FALSE;
	END_VAR
	VAR_OUTPUT
		/* See Section 5.1.2 General Output Parameters */
		Ready : BOOL := FALSE;
		/* Output for the safety-related response.
		 * FALSE: Safety output disabled. Demand for safety-related response (e.g., reset required or internal errors active).
		 * TRUE: Safety output enabled. No demand for safety-related response.
		 */
		S_ESPE_Out : SAFEBOOL := SAFEBOOL_Constant#SAFEFALSE;
		/* Optional. See 5.1.2 General Output Parameters */
		SafetyDemand : BOOL := FALSE;
		/* Optional. See 5.1.2 General Output Parameters */
		ResetRequest : BOOL := FALSE;
		/* See Section 5.1.2 General Output Parameters */
		Error : BOOL := FALSE;
		/* See Section 5.1.2 General Output Parameters */
		DiagCode : WORD := 16#0000;
	END_VAR
	VAR
		GenericSafetyDemand : SFB_GenericSafetyDemand;
	END_VAR

	GenericSafetyDemand(
		Activate := Activate,
		S_SafetyDemandIn := S_ESPE_In,
		S_StartReset := S_StartReset,
		S_AutoReset := S_AutoReset,
		Reset := Reset,
		Ready => Ready,
		S_SafetyDemandOut => S_ESPE_Out,
		SafetyDemand => SafetyDemand,
		ResetRequest => ResetRequest,
		Error => Error,
		DiagCode => DiagCode,
		ENO => ENO
	);

END_FUNCTION_BLOCK

END_NAMESPACE
END_NAMESPACE

(* ---- SF_Guard.iecst ---- *)
USING logicals.web.standard.safe;

NAMESPACE logicals.web.standard.safe
NAMESPACE plcopen

TYPE
	SF_Guard_State : UINT(
	/* Static reset detected in state 8003. */
	Reset_Error := 16#C001,
	/* DiscrepancyTime elapsed in state 8806. */
	Discrepancytime_Error_1 := 16#C010,
	/* DiscrepancyTime elapsed in state 8808. */
	Discrepancytime_Error_2 := 16#C020,
	/* The function block is not active (initial state). */
	Idle := 16#0000,
	/* Safety guard closed and Safe state acknowledged. */
	Normal := 16#8000,
	/* Function block has been activated. */
	Init := 16#8001,
	/* Complete switching sequence required. */
	Open_Guard_Request := 16#8802,
	/* Waiting for rising trigger at Reset. */
	Wait_For_Reset := 16#8402,
	/* Guard completely opened. */
	Guard_Opened := 16#8804,
	/* S_GuardSwitch1 has been switched to TRUE - waiting for S_GuardSwitch2; discrepancy timer started. */
	Wait_For_GuardSwitch2 := 16#8806,
	/* S_GuardSwitch2 has been switched to TRUE - waiting for S_GuardSwitch1; discrepancy timer started. */
	Wait_For_GuardSwitch1 := 16#8808,
	/* Guard closed. Waiting for Reset, if S_AutoReset = FALSE. */
	Guard_Closed := 16#8002
	);
END_TYPE

/*
 * This function block monitors the relevant safety guard.
 * There are two independent input parameters for two switches at the safety guard coupled with a time difference (DiscrepancyTime) for closing the guard.
 */
FUNCTION_BLOCK SF_Guard
	{ altName:="SF_Guard"; bgColor:="Gold"; width:=360; }
	VAR_INPUT
		/* See Section 5.1.1 General Input Parameters */
		Activate : BOOL := FALSE;
		/* Variable.
		 * Guard switch 1 input.
		 * FALSE: Guard is not closed.
		 * TRUE: Guard is closed. */
		S_GuardSwitch1 : SAFEBOOL := SAFEBOOL_Constant#SAFEFALSE;
		/* Variable.
		 * Guard switch 2 input.
		 * FALSE: Guard is not closed.
		 * TRUE: Guard is closed. */
		S_GuardSwitch2 : SAFEBOOL := SAFEBOOL_Constant#SAFEFALSE;
		/* Constant.
		 * Configures the monitored synchronous time between S_GuardSwitch1 and S_GuardSwitch2. */
		DiscrepancyTime : TIME := T#0ms;
		/* See Section 5.1.1 General Input Parameters */
		S_StartReset : SAFEBOOL := SAFEBOOL_Constant#SAFEFALSE;
		/* See Section 5.1.1 General Input Parameters */
		S_AutoReset : SAFEBOOL := SAFEBOOL_Constant#SAFEFALSE;
		/* See Section 5.1.1 General Input Parameters */
		 Reset : BOOL := FALSE;
	END_VAR

	VAR_OUTPUT
		/* See Section 5.1.2 General Output Parameters */
		Ready : BOOL := FALSE;
		/* Output indicating that the guard is closed and the guarded area safe
		 * FALSE: Guard is open.
		 * TRUE: both S_GuardSwitches are TRUE, no error and acknowledgment. Guard is closed.. */
		S_GuardOut : SAFEBOOL := SAFEBOOL_Constant#SAFEFALSE;
		/* See Section 5.1.2 General Output Parameters */
		SafetyDemand : BOOL := FALSE;
		/* See Section 5.1.2 General Output Parameters */
		ResetRequest : BOOL := FALSE;
		/* See Section 5.1.2 General Output Parameters */
		Error : BOOL := FALSE;
		/* See Section 5.1.2 General Output Parameters */
		DiagCode : WORD := 16#0000;
	END_VAR

	VAR
		DiscrepancyTimer : TON;
		R_Trig_Reset : R_TRIG;
	END_VAR

	R_Trig_Reset(Reset);

	IF(NOT Activate) THEN
		DiagCode := TO_WORD(SF_Equivalent_State#Idle);
	ELSE
		CASE TO_UINT(DiagCode) OF
			SF_Guard_State#Idle:
				/* IF(Activate) THEN - Active is always true here */
					DiagCode := TO_WORD(SF_Guard_State#Init);
			SF_Guard_State#Init:
				IF(IS_NOT(S_GuardSwitch1) OR IS_NOT(S_GuardSwitch2)) THEN
					DiagCode := TO_WORD(SF_Guard_State#Open_Guard_Request);
				ELSIF(IS(S_GuardSwitch1) AND IS(S_GuardSwitch2) AND IS_NOT(S_StartReset)) THEN
					DiagCode := TO_WORD(SF_Guard_State#Wait_For_Reset);
				/*ELSIF(IS(S_GuardSwitch1) AND IS(S_GuardSwitch2) AND IS(S_StartReset)) THEN - S_GuardSwitch1 and S_GuardSwitch2 can only be true here, S_StartReset can only be true */
				ELSE
					DiagCode := TO_WORD(SF_Guard_State#Normal);
				END_IF;
			SF_Guard_State#Open_Guard_Request:
				IF(IS_NOT(S_GuardSwitch1) AND IS_NOT(S_GuardSwitch2)) THEN
					DiagCode := TO_WORD(SF_Guard_State#Guard_Opened);
				END_IF;
			SF_Guard_State#Guard_Opened:
				IF(IS(S_GuardSwitch1)) THEN
					DiagCode := TO_WORD(SF_Guard_State#Wait_For_GuardSwitch2);
				ELSIF(IS(S_GuardSwitch2)) THEN
					DiagCode := TO_WORD(SF_Guard_State#Wait_For_GuardSwitch1);
				END_IF;
			SF_Guard_State#Wait_For_GuardSwitch2:
				DiscrepancyTimer();
				IF(DiscrepancyTimer.Q) THEN
					DiagCode := TO_WORD(SF_Guard_State#Discrepancytime_Error_1);
				ELSIF(IS_NOT(S_GuardSwitch1)) THEN
					DiagCode := TO_WORD(SF_Guard_State#Open_Guard_Request);
				ELSIF(IS(S_GuardSwitch1) AND IS(S_GuardSwitch2)) THEN
					DiagCode := TO_WORD(SF_Guard_State#Guard_Closed);
				END_IF;
			SF_Guard_State#Wait_For_GuardSwitch1:
				DiscrepancyTimer();
				IF(DiscrepancyTimer.Q) THEN
					DiagCode := TO_WORD(SF_Guard_State#Discrepancytime_Error_2);
				ELSIF(IS_NOT(S_GuardSwitch2)) THEN
					DiagCode := TO_WORD(SF_Guard_State#Open_Guard_Request);
				ELSIF(IS(S_GuardSwitch1) AND IS(S_GuardSwitch2)) THEN
					DiagCode := TO_WORD(SF_Guard_State#Guard_Closed);
				END_IF;
			SF_Guard_State#Discrepancytime_Error_1,
			SF_Guard_State#Discrepancytime_Error_2:
				IF(IS_NOT(S_GuardSwitch1) AND IS_NOT(S_GuardSwitch2)) THEN
					DiagCode := TO_WORD(SF_Guard_State#Guard_Opened);
				END_IF;
			SF_Guard_State#Guard_Closed:
				IF(IS_NOT(S_GuardSwitch1) OR IS_NOT(S_GuardSwitch2)) THEN
					DiagCode := TO_WORD(SF_Guard_State#Open_Guard_Request);
				ELSIF(IS_NOT(S_AutoReset)) THEN
					DiagCode := TO_WORD(SF_Guard_State#Wait_For_Reset);
				/* ELSIF(IS(S_AutoReset)) THEN - S_AutoReset can only be true here */
				ELSE
					DiagCode := TO_WORD(SF_Guard_State#Normal);
				END_IF;
			SF_Guard_State#Wait_For_Reset:
				IF(Reset AND NOT R_Trig_Reset.Q) THEN
					DiagCode := TO_WORD(SF_Guard_State#Reset_Error);
				ELSIF(IS_NOT(S_GuardSwitch1) OR IS_NOT(S_GuardSwitch2)) THEN
					DiagCode := TO_WORD(SF_Guard_State#Open_Guard_Request);
				ELSIF(R_Trig_Reset.Q) THEN
					DiagCode := TO_WORD(SF_Guard_State#Normal);
				END_IF;
			SF_Guard_State#Normal:
				IF(IS_NOT(S_GuardSwitch1) OR IS_NOT(S_GuardSwitch2)) THEN
					DiagCode := TO_WORD(SF_Guard_State#Open_Guard_Request);
				END_IF;
			SF_Guard_State#Reset_Error:
				IF(NOT Reset) THEN
					DiagCode := TO_WORD(SF_Guard_State#Wait_For_Reset);
				END_IF;
		END_CASE;
	END_IF;

	CASE TO_UINT(DiagCode) OF
		SF_Guard_State#Idle:
			DiscrepancyTimer(IN := FALSE);
			Ready := FALSE;
			S_GuardOut := SAFEBOOL_Constant#SAFEFALSE;
			SafetyDemand := FALSE;
			ResetRequest := FALSE;
			Error := FALSE;
		SF_Guard_State#Normal:
			DiscrepancyTimer(IN := FALSE);
			Ready := TRUE;
			S_GuardOut := SAFEBOOL_Constant#SAFETRUE;
			SafetyDemand := FALSE;
			ResetRequest := FALSE;
			Error := FALSE;
		SF_Guard_State#Init,
		SF_Guard_State#Guard_Closed:
			DiscrepancyTimer(IN := FALSE);
			Ready := TRUE;
			S_GuardOut := SAFEBOOL_Constant#SAFEFALSE;
			SafetyDemand := FALSE;
			ResetRequest := FALSE;
			Error := FALSE;
		SF_Guard_State#Open_Guard_Request,
		SF_Guard_State#Guard_Opened:
			DiscrepancyTimer(IN := FALSE);
			Ready := TRUE;
			S_GuardOut := SAFEBOOL_Constant#SAFEFALSE;
			SafetyDemand := TRUE;
			ResetRequest := FALSE;
			Error := FALSE;
		SF_Guard_State#Wait_For_GuardSwitch2,
		SF_Guard_State#Wait_For_GuardSwitch1:
			DiscrepancyTimer(IN := TRUE, PT := DiscrepancyTime);
			Ready := TRUE;
			S_GuardOut := SAFEBOOL_Constant#SAFEFALSE;
			SafetyDemand := TRUE;
			ResetRequest := FALSE;
			Error := FALSE;
		SF_Guard_State#Wait_For_Reset:
			DiscrepancyTimer(IN := FALSE);
			Ready := TRUE;
			S_GuardOut := SAFEBOOL_Constant#SAFEFALSE;
			SafetyDemand := FALSE;
			ResetRequest := TRUE;
			Error := FALSE;
		SF_Guard_State#Reset_Error,
		SF_Guard_State#Discrepancytime_Error_1,
		SF_Guard_State#Discrepancytime_Error_2:
			DiscrepancyTimer(IN := FALSE);
			Ready := TRUE;
			S_GuardOut := SAFEBOOL_Constant#SAFEFALSE;
			SafetyDemand := FALSE;
			ResetRequest := FALSE;
			Error := TRUE;
		ELSE
			ENO := FALSE;
	END_CASE;

	ENO := ENO AND CheckSAFEBOOL(S_GuardSwitch1) AND CheckSAFEBOOL(S_GuardSwitch2) AND CheckSAFEBOOL(S_StartReset) AND CheckSAFEBOOL(S_AutoReset);

END_FUNCTION_BLOCK

END_NAMESPACE
END_NAMESPACE
